FUNCTION_BLOCK "GCS7_E_FBAL"	// FB 28
TITLE = MZAG/MZAH/MZDE Flowbalancer
//  
//COPYRIGHT:    (C) 1997 BY  BUHLER AG, CH-9240 UZWIL  SWITZERLAND
//
//PRODUCT:      GCS7
//
//TITLE:        Element MZAG/MZAH/FBAL,MZDE (Profibus and Opto22)
//              (GCPROVB Revision 11)
//
//-------------------------------------------------------------------------
//
//IDENT:        AUTHOR:             DEPT:                      DATE:
//FB28.7.6      A. Egli             BASE                       30-Oct-2008
//              - StStopping -->StStopped : Check LCStep<=2
//FB28.7.5      A. Egli             BASE                       12-Jun-2008
//              - Disable Alarm26 if InRestdischarge=True
//FB28.7.4      A. Egli             BASE                       09-Apr-2008
//              Disable Alarm 18 Battery Low
//FB28.7.3      A. Egli             CT3                        08-Apr-2008
//              - Remove StStopping -->StStarting 
//              - StStopping -->StStopped : Check LCStep=1
//              - Filter.A34NoProduct and A37Empty catched until stopped
//FB28.7.2      A. Egli             CT3                        25-Mai-2007
//              - Overflow weight OutNotErasableWeight is 999'999'999 
//FB28.7.1      A.Egli              CT3                        01-Dec-2005
//              Parameter Upload Change DBD86-->DBD88
//FB28.7.0      A.Egli              CT3                        05-Jan-2005
//              Parameter Upload (uses DB10)
//FB28.6.0      A.Egli              CT3                        17-Aug-2004
//              MZDE: InRestdicharge
//FB28.5.3      A.Egli              CT3                        13-Apr-2004
//              MZDE: Reset "CmdNewJob"
//FB28.5.2      A.Egli              CT3                        17-Nov-2003
//              - Alarm 90: Fault Remote Control
//              - Ignor SumFault as long AlarmNr <> 0
//              - ComFault in mocal mode: change to StStopped 
//FB28.5.1      A. Egli             CT3                        11-Nov-2003
//              - No restart during StStopping.
//FB28.5.0      A. Egli             CT3                        09-Sep-2003
//              - ParMZDE 
//              - Condition for stoppen when stop point is reached 
//FB28.4.0      A. Egli             CT3                        17-Jun-2002
//              - New Release with one block 
//              - Profibus and Opto22 
//              - MZMN Micro Dosing
//              - LC Alarm 14 (DPFault) =Log Text number 12
//              - Command A: Command Flowrate in %
//FB28.3.1      A. Egli             CT3                        11-Jul-2000
//              MZAH mode: Command A, h
//FB28.3.0      A. Egli             CT3                        20-Jun-2000
//              Automatic set zero point
//FB28.2.2      A. Egli             CT3                        17-Mar-2000
//              Length for answer telegram
//FB33.2B       A. Egli             CT3                        20-Juli-1999
//              No fault is element InLocal
//FB33.2A       S. Kalberer         CT3                        11-Mar-1999
//              Correction factor ('K') included
//              CmdNewJob sets CmdNewValue
//FB33.1A       A. Egli             CT3                        16-Apr-1998
//              1st Release in S7
//
//-------------------------------------------------------------------------
//
//PURPOSE:      MANUAL : see [MZAHxxMAN]
//
//RESTRICTIONS: S7
//
//              (*2) : Not used for MZDE
//
//=======================================================
//Log Message: 
//------------------------------------------------------
//0     = Fault Cannceled
//1..79 = AlarmLC : Alarmnumber see manual of MEAF
//90    = Fault Remote Control
//91    = StStopped
//92    = StDosing
//93    = StEmptied
//94    = Timeout starting
//95    = Wrong value
//96    = Communication fault
//97    = 
//98    = 
//99    = Collected alarm
//
//=======================================================
//StCode:  State               
//------------------------------------------------------
//32    StFault                 
// 1    StStopped                   Stopped
//41    Stopped.HWStop              StStopped + InHWStop 
//51    Stopped.DPFault             StStopped + DPFault
// 2    StStarting              
// 3    StStarted               
// 7    StStopping              
//
//
AUTHOR : EA
FAMILY : GCS7LL
NAME : FBAL
VERSION : 7.6
VAR
  StCode : INT ;	//Element state code
  InEnable : BOOL ;	//Enable to run the element (manual and automatic mode)
  InRestdischarge : BOOL ;	//Rest discharge of the bin
  spare22 : BOOL ;
  CmdSetZeroPoint : BOOL ;	//Set zero point (*2)
  CmdNewValue : BOOL ;	//Send new target values
  CmdNewJob : BOOL ;	//Clear actual values (*2)
  CmdCorrFactor : BOOL ;	//Set correction factor (*2)
  tmpFilter34_37 : BOOL ;
  CmdOff : BOOL ;	//Pulse to stop the element (manual mode)
  CmdOn : BOOL ;	//Pulse to start the element (manual mode)
  CmdNext : BOOL ;	//Pulse to start the element in automatic mode
  CmdFaultReset : BOOL ;	//Command to reset fault
  InLocal : BOOL ;	//1= Local mode (no fault by start with service switch)
  InManual : BOOL ;	//1= Manual / 0= Automatic
  InReport : BOOL ;	//Report of all state transitions
  spare0307 : BOOL ;
  InHWStop : BOOL ;	//HW stop is detected, no fault
  InDPFault : BOOL ;	//DP-Fault is detected, no fault
  InSimulation : BOOL ;	//MZAH: Simulation with DPSim
  OutComFault : BOOL ;	//Communication fault
  OutBinEmpty : BOOL ;	//FBAL is rest discharged (*2)
  OutSetZeroPoint : BOOL ;	//(*2)
  OutSystemAdjust : BOOL ;	//(*2)
  OutpDosingEnable : BOOL ;	//Digital output dosing enable (only Opto22)
  StStopped : BOOL ;	//Element is stopped
  StStarting : BOOL ;	//Element is starting
  StStarted : BOOL ;	//Element is dosing
  StStopping : BOOL ;	//Element is stopping
  StFault : BOOL ;	//Element has a communication or device fault
  spare55 : BOOL ;
  spare56 : BOOL ;
  spare57 : BOOL ;
  OutStopPoint : BOOL ;	//Target weight reached (*2)
  OutWrongValue : BOOL ;	//Wrong nominal values, rejected by MEAF
  InFlowrate : DINT ;	//Flowrate target value [0.1%] or [kg/h] ! MZDE:Position [0.1%]
  InJobWeight : DINT ;	//MZAH: Is send to LC (*2)
  InRecipeNr : INT ;	//MZAH: Is send to LC (*2)
  InCorrFactor : DINT  := L#1000;	//Correction factor (1000: neutral value = no correction) (*2)
  OutFlowrate : DINT ;	//Is read from LC  FBAL:[kg/h]  ! MZDE:Position [0.1%]
  OutJobWeight : DINT ;	//Is calculated by element out of the not erasable weight  (*2)
  OutTotalWeight : DINT ;	//Is read from LC: de: Totalgewicht (*2)
  OutScaleWeight : DINT ;	//Is read from LC
  OutSetZeroTime : INT ;	//Actual time to set zero point (*2)
  OutRecipeNr : INT ;	//Is read from MEAF (*2)
  OutLCStep : INT ;	//Is read from MEAF
  OutAlarmNr : INT ;	//Is read from MEAF
  OutAlarmNrLog : INT ;	//Last textnumber send to log
  Par : STRUCT
   ParObjectNo : INT ;	//Is used for communication with PC, e.g. for message
   ParMsgType : INT ;	//Is used for message (translation of state)
   ParHornCode : INT ;	//Is used by horn module
   ParLogOff : BOOL ;	//Report is off
   ParManual : BOOL ;	//Manual mode wihout interlocking
   ParWithFlowratePc : BOOL ;	//Target flowrate in 0.1 %
   ParMZAH : BOOL ;	//MZAH Mode
   ParOpto22 : BOOL ;	//1=OPTO22 communication, 0=DP
   ParMZDE : BOOL ;	//MZDE ELement
   ParFilter : STRUCT 	//Filter to alarm 1=Ignore alarm
    SumFault : BOOL ;	//All: de: Sammelalarm
    A05_24VToLow : BOOL ;	//All:
    A07ADRange : BOOL ;
    A08ADCalibration : BOOL ;
    A09ADFunction : BOOL ;
    A10ADSupply : BOOL ;
    A11AnalogInput : BOOL ;
    AxxCommunication : BOOL ;	//A12: Serial Interface ; A14=DPFault
    A13RemoteControl : BOOL ;
    A16Printer : BOOL ;
    A24WeightHopper : BOOL ;
    A25FrequenceConverter : BOOL ;
    A26Tolerance : BOOL ;
    A27Measurment : BOOL ;
    A28Feeddrive : BOOL ;
    A29FeedingTime : BOOL ;
    A30ZeroTara : BOOL ;	//MZAH
    A32InletSlideGate : BOOL ;	//MZAH
    A33AirPressure : BOOL ;	//MZAH
    A34NoProduct : BOOL ;
    A37Empty : BOOL ;	//MZAH
    A38Slide : BOOL ;	//MZAH
    A39AirPressure : BOOL ;	//MZAH
    A54Relais : BOOL ;	//MZMN
   END_STRUCT ;
   ParComDB : INT ;	//OPTO22  : Communication DB
   ParLCIdx : INT ;	//OPTO22  : Index of data record
   ParLCAddr : INT ;	//OPTO22  : Address of LC
   ParIOByteNr : INT ;	//PROFIBUS: Address of first input and output byte
   ParMonTime : INT ;	//Monitoring time starting and stopping
   OutMonTime : INT ;	//Monitoring time starting and stopping
   OutNotErasableWeight : DINT  := L#-1;	//Is read from FBAL
   OutHelpFlags : STRUCT 	//Is sent to FBAL
    OutAlarmTimeOut : BOOL ;
    CmdNewValue : BOOL ;
    CmdFaultReset : BOOL ;
    CmdNewJob : BOOL ;
    OutFaultResetDone : BOOL ;
    OutTestNewAlarm : BOOL ;	//Aux. signal to retry fault message
    CmdCorrFactor : BOOL ;
    spare0007 : BOOL ;
    OutRelevantFault : BOOL ;
    OutNoAlarm : BOOL ;	//Alarmnumber 0 is read form LC
    OutFlagFaultResetDone : BOOL ;
    OutWeightCleared : BOOL ;	//Erasable weight is cleared
    OutComFaultRead : BOOL ;
    OutComFaultSend : BOOL ;
   END_STRUCT ;
   Command : STRUCT
    Start : BOOL ;	//de: Start
    ResetWtTotal : BOOL ;	//FBAL: de: Total löschen (*2)
    Restdischarge : BOOL ;	//MZDE: de: Restentleeren
    spare03 : BOOL ;
    spare04 : BOOL ;
    OverwriteLL : BOOL ;	//FBAL: de: Kein Alarm bei Leerstand (*2)
    spare06 : BOOL ;
    AcceptNewDataReady : BOOL ;	//FBAL: de: Quittierung neue Werte Bereit
    spare10 : BYTE ;
    spare20 : BYTE ;
    CommandReady : BOOL ;	//de: Steuersignale gültig
    SetZeroPoint : BOOL ;	//MZAG: de: MZAG (*2)
    spare32 : BOOL ;
    spare33 : BOOL ;
    spare34 : BOOL ;
    ResetAlarm : BOOL ;	//de: Alarm löschen
    NewSendData : BOOL ;	//de: Aenderung Sendedaten
    AcceptNewRcvData : BOOL ;	//de: Quittierung Aenderung Empfangsdatensatz
   END_STRUCT ;
   Status : STRUCT
    Operation : BOOL ;	//de: Betrieb
    WtTotalReached_InPos : BOOL ;	//de: Total erreicht  : MZDE: Slide in position
    RestdischargeDone : BOOL ;	//MZDE: de: Restentleeren ausgeführt
    spare03 : BOOL ;
    TotalReady : BOOL ;	//de: Total bereit (*2)
    Empty : BOOL ;	//de: Silo leer (*2)
    WtPulse : BOOL ;	//de: Gewichtsimpuls (*2)
    NewDataReady : BOOL ;	//de: Neue Werte Bereit
    AnalogMode : BOOL ;	//0/4-20mA set value  (*2)
    SetZeroPoint_Recipe1 : BOOL ;	//(*2)
    SystemAdjust_Recipe2 : BOOL ;	//(*2)
    spare20 : BYTE ;
    spare30 : BOOL ;
    spare31 : BOOL ;
    spare32 : BOOL ;
    RemoteControl : BOOL ;	//de: Sollwertvorgabe Remote
    WrongValue : BOOL ;	//de: Falscher Sollwert
    SumFault : BOOL ;	//de: Sammelalarm
    AcceptNewSendData : BOOL ;	//de: Quittierung Aenderung Sendedaten
    NewRcvData : BOOL ;	//de: Aenderung Empfangsdaten
   END_STRUCT ;
   OutComFlags : STRUCT 	//Flags for communication
    i_Done : BOOL ;
    d_Done : BOOL ;
    h_done : BOOL ;
    Q_Done : BOOL ;
    P_Done : BOOL ;
    S_Done : BOOL ;
    K_Done : BOOL ;
    A_Done : BOOL ;
   END_STRUCT ;
  END_STRUCT ;
END_VAR
VAR_TEMP
  tmpLOGvalue : WORD ;	//LOG value
  tmpCommand : INT ;
  tmpFBNO : INT ;	//Number of the actual FB
  tmpFault : BOOL ;
  tmpOff : BOOL ;
  tmpOn : BOOL ;
  tmpLocal : BOOL ;
  tmpLocalFault : BOOL ;
  tmpReport : BOOL ;
  tmpFlag : BOOL ;
  tmpOutLCAlarmBinEmpty : BOOL ;
  tmpLenDyn : DINT ;
  tmpWt : DINT ;
  tmpFilter : ARRAY  [0 .. 100 ] OF BOOL ;
  tmpComDB : INT ;
  tmpStatus_h : STRUCT 	//Is read from FBAL
   Remote : BOOL ;
   NewValue : BOOL ;
   Z1_Bit2 : BOOL ;
   BinEmpty : BOOL ;
   Z2_Bit0 : BOOL ;
   Z2_Bit1 : BOOL ;
   Z2_Bit2 : BOOL ;
   SumFault : BOOL ;
  END_STRUCT ;
  tmpStatus_i : STRUCT 	//Is read from FBAL
   EnableInactive : BOOL ;
   AlarmActive : BOOL ;
   AnalogMode : BOOL ;	//0/4-20mA set value
   SetZeroPoint : BOOL ;
   SystemAdjust : BOOL ;
   spare15 : BOOL ;	//only MEAF
   spare16 : BOOL ;	//only MEAF
   NominalFailure : BOOL ;	//Nominal value < 1%
  END_STRUCT ;
  tmpCommand_A : STRUCT
   Start : BOOL ;
   Stop : BOOL ;
   ResetWtTotal : BOOL ;
   AlarmReset : BOOL ;
   ValueInPc : BOOL ;
   Z3_1 : BOOL ;
   Z3_2 : BOOL ;
   Modify : BOOL ;
  END_STRUCT ;
  tmpCommand_S : STRUCT
   SetDosingRelease : BOOL ;
   AlarmReset : BOOL ;
   spare16 : BOOL ;
   SetZeroPoint : BOOL ;
   ClearPowerFlag : BOOL ;
   ResetWtTotal : BOOL ;
   spare12 : BOOL ;
   spare13 : BOOL ;
  END_STRUCT ;
  tmpAddr : WORD ;
  tmpReturn : INT ;
  DPData : STRUCT
   StatusCommand : DWORD ;
   NrSndDataSet : BYTE ;	//de: Nummer Sendedatensatz
   IdxSndDataSet : BYTE ;	//de: Index Sendedatensatz
   NrRcvDataSet : BYTE ;	//de: Nummer Empfangsdatensatz
   IdxRcvDataSet : BYTE ;	//de: Index Empfangsdatensatz
   Data : ARRAY  [1 .. 4 ] OF DINT ;
  END_STRUCT ;
  Set001 : STRUCT
   FlowrateAc : DINT ;	//de: Istleistung kg/h
   WtTotalAc : DINT ;	//de: Isttotalgewicht kg
   WtNotErasable : DINT ;	//de: nochtlöschbarese Totalgewicht
   spare12 : BYTE ;
   RecipeNr : BYTE ;
   Step : BYTE ;
   AlarmNr : BYTE ;
  END_STRUCT ;
END_VAR
BEGIN
NETWORK
TITLE =  Start Global
      L     28;
      T     #tmpFBNO;
      L     88;
      T     #tmpLenDyn;	//--> Len dynamic data in byte
      L     #Par.ParComDB;
      T     #tmpComDB;
NETWORK
TITLE = Filter
      LAR1  P##tmpFilter;
      L     0;
      T     LD [AR1,P#0.0];	//tmpFilter[00..31]  //[5.0]
      T     LD [AR1,P#4.0];	//tmpFilter[32..63]  //[5.0]
      T     LD [AR1,P#8.0];	//tmpFilter[64..95]  //[5.0]
      SET;	//[5.2]
      =     #tmpFilter[0];
      A     #Par.ParFilter.A05_24VToLow;
      =     #tmpFilter[5];
      A     #Par.ParFilter.A07ADRange;
      =     #tmpFilter[7];
      A     #Par.ParFilter.A08ADCalibration;
      =     #tmpFilter[8];
      A     #Par.ParFilter.A09ADFunction;
      =     #tmpFilter[9];
      A     #Par.ParFilter.A10ADSupply;
      =     #tmpFilter[10];
      A     #Par.ParFilter.A11AnalogInput;
      =     #tmpFilter[11];
      A     #Par.ParFilter.AxxCommunication;
      =     #tmpFilter[12];
      =     #tmpFilter[14];	//[1.4]
      A     #Par.ParFilter.A13RemoteControl;
      =     #tmpFilter[13];
      A     #Par.ParFilter.A16Printer;
      =     #tmpFilter[16];
      SET;
      =     #tmpFilter[18];	//[7.4] Battery Low
      A     #Par.ParFilter.A24WeightHopper;
      =     #tmpFilter[24];
      A     #Par.ParFilter.A25FrequenceConverter;
      =     #tmpFilter[25];
      A     #Par.ParFilter.A26Tolerance;
      O     #InRestdischarge;	//[7.5]
      =     #tmpFilter[26];
      A     #Par.ParFilter.A27Measurment;
      =     #tmpFilter[27];
      A     #Par.ParFilter.A28Feeddrive;
      =     #tmpFilter[28];
      A     #Par.ParFilter.A29FeedingTime;
      =     #tmpFilter[29];
      A     #Par.ParFilter.A30ZeroTara;
      =     #tmpFilter[30];
      A     #Par.ParFilter.A32InletSlideGate;
      =     #tmpFilter[32];
      A     #Par.ParFilter.A33AirPressure;
      =     #tmpFilter[33];
      A     #InRestdischarge;	//[7.3]
      S     #tmpFilter34_37;	//[7.3]
      A     #StStopped;	//[7.3]
      R     #tmpFilter34_37;	//[7.3]
      A     #tmpFilter34_37;	//[7.3]
      A     #StStopping;	//[7.3]
      O     #Par.ParFilter.A34NoProduct;
      O     #InRestdischarge;
      =     #tmpFilter[34];
      A     #tmpFilter34_37;	//[7.3]
      A     #StStopping;	//[7.3]
      O     #Par.ParFilter.A37Empty;
      O     #InRestdischarge;
      =     #tmpFilter[37];
      A     #Par.ParFilter.A38Slide;
      =     #tmpFilter[38];
      A     #Par.ParFilter.A39AirPressure;
      =     #tmpFilter[39];
      A     #Par.ParFilter.A54Relais;
      =     #tmpFilter[54];
NETWORK
TITLE = (Opto22) Call back function
//*****This functions are called by FBxxx (COM) ******
      AN    #Par.ParOpto22;
      JC    O22Z;
      OPN   DB [#tmpComDB];
      L     0;
      L     DBW 32;	//COM.Element.CODE;
      ==I;
      JC    PC;
      L     DBB 76;	//COM.Telegram.Command;
      T     #tmpCommand;
      L     1;
      L     DBW 32;	//COM.Element.CODE;
      ==I;
      JC    Send;
      L     2;
      ==I;
      JC    Rcv;
      L     4;	//NAK
      L     DBW 32;	//COM.Element.CODE;
      ==I;
      S     #OutComFault;	//fault communication
      JU    STOR;
//Read telegram length
Send: L     #tmpCommand;
      L     'd';
      ==I;
      L     16;	//Lenght in byte
      JC    Sndx;
      L     #tmpCommand;
      L     'i';
      ==I;
      L     6;	//Lenght in byte
      JC    Sndx;
      L     #tmpCommand;
      L     'h';
      ==I;
      L     36;	//Lenght in byte
      JC    Sndx;
      JU    SndW;
Sndx: T     DBW 86;	//COM.Telegram.LenAnswer
      JU    STOR;
SndW: NOP   0;
//======================================================================
//Prepare Send Data 
//======================================================================
//--------------------
//Send Q
//--------------------
      L     #tmpCommand;
      L     'Q';
      <>I;
      JC    SndP;
      L     #InFlowrate;
      T     DBD 36;	//COM.Element.InOutValue
      L     16;	//Convert DInt to 6-ASCII
      T     DBW 0;	//COM.CODE
      L     6;	//Lenght in byte
      JU    Snd1;
//--------------------
//Send P
//--------------------
SndP: L     #tmpCommand;
      L     'P';
      <>I;
      JC    SndK;
      L     #InFlowrate;
      T     DBD 36;	//COM.Element.InOutValue
      L     14;	//Convert DInt to 4-ASCII
      T     DBW 0;	//COM.CODE
      L     4;	//Lenght in byte
      JU    Snd1;
//--------------------
//Send K [2.A]
//--------------------
SndK: L     #tmpCommand;
      L     'K';
      <>I;
      JC    SndA;
      L     #InCorrFactor;
      T     DBD 36;	//COM.Element.InOutValue
      L     16;	//Convert DInt to 6-ASCII
      T     DBW 0;	//COM.CODE
      L     6;	//Lenght in byte
      JU    Snd1;
//--------------------
//Send A [3.1]
//--------------------
SndA: L     #tmpCommand;
      L     'A';
      <>I;
      JC    SndS;
      LAR1  P##tmpCommand_A;
      L     0;
      T     LW [AR1,P#0.0];	//-->Reset tmpStateTarget
//command 1
      A     #Par.Command.Start;
      =     #tmpCommand_A.Start;
      AN    #Par.Command.Start;
      =     #tmpCommand_A.Stop;
      A     #Par.Command.ResetWtTotal;
      =     #tmpCommand_A.ResetWtTotal;
      A     #Par.Command.ResetAlarm;
      =     #tmpCommand_A.AlarmReset;
      A     #Par.ParWithFlowratePc;	//[4.0]
      =     #tmpCommand_A.ValueInPc;	//[4.0]
      SET;
      =     #tmpCommand_A.Modify;
      L     0;	//Character offset
      T     DBW 40;	//COM.Element.AddrOffset
      LAR1  P##tmpCommand_A;
      L     LB [AR1,P#0.0];
      T     DBD 36;	//COM.Element.InOutValue
      L     31;	//Convert Hex to 1-ASCII
      T     DBW 0;	//COM.CODE
      CDB;	//ComDB->Instanz-DB
      UC    "GCS7_RS485Ctrl";	//Convert (CODE=DBW0)
      CDB;	//ElementDB->Instanz-DB
//n.b   
      L     1;	//Character offset
      T     DBW 40;	//COM.Element.AddrOffset
      L     0;
      T     DBD 36;	//COM.Element.InOutValue
      L     32;	//Convert Hex to 1-ASCII
      T     DBW 0;	//COM.CODE
      CDB;	//ComDB->Instanz-DB
      UC    "GCS7_RS485Ctrl";	//Convert (CODE=DBW0)
      CDB;	//ElementDB->Instanz-DB
// Command 2    
      L     3;	//Character offset
      T     DBW 40;	//COM.Element.AddrOffset
      LAR1  P##tmpCommand_A;
      L     LB [AR1,P#0.0];
      SRW   4;
      T     DBD 36;	//COM.Element.InOutValue
      L     31;	//Convert Hex to 1-ASCII
      T     DBW 0;	//COM.CODE
      CDB;	//ComDB->Instanz-DB
      UC    "GCS7_RS485Ctrl";	//Convert (CODE=DBW0)
      CDB;	//ElementDB->Instanz-DB
// n.b    
      L     4;	//Character offset
      T     DBW 40;	//COM.Element.AddrOffset
      L     0;
      T     DBD 36;	//COM.Element.InOutValue
      L     16;	//Convert DInt to 6-ASCII
      T     DBW 0;	//COM.CODE
      CDB;	//ComDB->Instanz-DB
      UC    "GCS7_RS485Ctrl";	//Convert (CODE=DBW0)
      CDB;	//ElementDB->Instanz-DB
// Flowrate    
      L     6;	//Character offset
      T     DBW 40;	//COM.Element.AddrOffset
      L     #InFlowrate;
      T     DBD 36;	//COM.Element.InOutValue
      L     16;	//Convert DInt to 6-ASCII
      T     DBW 0;	//COM.CODE
      CDB;	//ComDB->Instanz-DB
      UC    "GCS7_RS485Ctrl";	//Convert (CODE=DBW0)
      CDB;	//ElementDB->Instanz-DB
// InJobWeight                          //[5.0]
      L     12;	//Character offset
      T     DBW 40;	//COM.Element.AddrOffset
      L     #InJobWeight;
      T     DBD 36;	//COM.Element.InOutValue
      L     18;	//Convert DInt to 8-ASCII
      T     DBW 0;	//COM.CODE
      CDB;	//ComDB->Instanz-DB
      UC    "GCS7_RS485Ctrl";	//Convert (CODE=DBW0)
      CDB;	//ElementDB->Instanz-DB
      L     20;	//Lenght in byte
      T     DBW 78;	//COM.Telegram.Len
      JU    SndZ;
//--------------------
//Send S
//--------------------
SndS: L     #tmpCommand;
      L     'S';
      <>I;
      JC    SndZ;
      LAR1  P##tmpCommand_S;
      L     0;
      T     LW [AR1,P#0.0];	//-->Reset tmpStateTarget
      A     #Par.Command.Start;
      =     #tmpCommand_S.SetDosingRelease;
      A     #Par.Command.ResetAlarm;
      =     #tmpCommand_S.AlarmReset;
      =     #tmpCommand_S.ClearPowerFlag;
      A     #Par.Command.SetZeroPoint;
      =     #tmpCommand_S.SetZeroPoint;
      A     #Par.Command.ResetWtTotal;
      =     #tmpCommand_S.ResetWtTotal;
      LAR1  P##tmpCommand_S;
      L     LB [AR1,P#0.0];
      T     DBD 36;	//COM.Element.InOutValue
      L     32;	//Convert Hex to 2-ASCII
      T     DBW 0;	//COM.CODE
      L     2;	//Lenght in byte
Snd1: T     DBW 78;	//COM.Telegram.Len
      CDB;	//ComDB->Instanz-DB
      UC    "GCS7_RS485Ctrl";	//Convert (CODE=DBW0)
      CDB;	//ElementDB->Instanz-DB
SndZ: JU    STOR;
//======================================================================
//Answer Telegramm: Copy reveived data to element
//======================================================================
//--------------------
//Receive h 
//--------------------
Rcv:  R     #OutComFault;
      L     #tmpCommand;
      L     'h';
      <>I;
      JC    Rcvi;
      AN    #Par.OutHelpFlags.OutFaultResetDone;
      JC    r_H1;
      S     #Par.OutHelpFlags.OutTestNewAlarm;
//StepNr
r_H1: L     2;	//Character offset
      T     DBW 40;	//COM.Element.AddrOffset
      L     22;	//Convert 2-ASCII to DInt
      T     DBW 0;	//COM.CODE
      CDB;	//ComDB->Instanz-DB
      UC    "GCS7_RS485Ctrl";	//Convert (CODE=DBW0)
      CDB;	//ElementDB->Instanz-DB
      L     DBD 36;	//COM.Element.InOutValue
      T     #OutLCStep;
//LC status
      L     0;	//Character offset
      T     DBW 40;	//COM.Element.AddrOffset
      L     42;	//Convert 2-ASCII to Hex
      T     DBW 0;	//COM.CODE
      CDB;	//ComDB->Instanz-DB
      UC    "GCS7_RS485Ctrl";	//Convert (CODE=DBW0)
      CDB;	//ElementDB->Instanz-DB
      L     DBD 36;	//COM.Element.InOutValue
      LAR1  P##tmpStatus_h;
      T     LB [AR1,P#0.0];	//-->tmpStatus_h
      A     #tmpStatus_h.Remote;
      =     #Par.Status.RemoteControl;
      A     #tmpStatus_h.BinEmpty;
      =     #Par.Status.Empty;
      A     #tmpStatus_h.SumFault;
      =     #Par.Status.SumFault;
      L     #OutLCStep;
      L     3;
      >=I;
      =     #Par.Status.Operation;
      L     2;
      L     #OutLCStep;
      ==I;
      =     #Par.Status.SetZeroPoint_Recipe1;
//Alarm number / LC alarm bit mask
      L     4;	//Character offset
      T     DBW 40;	//COM.Element.AddrOffset
      L     22;	//Convert 2-ASCII to DInt
      T     DBW 0;	//COM.CODE
      CDB;	//ComDB->Instanz-DB
      UC    "GCS7_RS485Ctrl";	//Convert (CODE=DBW0)
      CDB;	//ElementDB->Instanz-DB
      L     DBD 36;	//COM.Element.InOutValue
      T     #OutAlarmNr;
//Filter SumFault
      L     #OutAlarmNr;	//[5.2]
      L     0;	//[5.2]
      <>I;	//[5.2]
      O     #Par.ParFilter.SumFault;	//[5.2]
      O     #InRestdischarge;	//[5.2]
      =     #tmpFilter[0];	//[5.2]
//Acutal flowrate
      L     6;	//Character offset
      T     DBW 40;	//COM.Element.AddrOffset
      L     26;	//Convert 6-ASCII to DInt
      T     DBW 0;	//COM.CODE
      CDB;	//ComDB->Instanz-DB
      UC    "GCS7_RS485Ctrl";	//Convert (CODE=DBW0)
      CDB;	//ElementDB->Instanz-DB
      L     DBD 36;	//COM.Element.InOutValue
      T     #OutFlowrate;
//ScaleWeight
      L     12;	//Character offset
      T     DBW 40;	//COM.Element.AddrOffset
      L     26;	//Convert 6-ASCII to DInt
      T     DBW 0;	//ERH.CODE
      CDB;	//ComDB->Instanz-DB
      UC    "GCS7_RS485Ctrl";	//Convert (CODE=DBW0)
      CDB;	//ElementDB->Instanz-DB
      L     DBD 36;	//ERH.Element.InOutValue
      T     #OutScaleWeight;	//[4.0]
//- OutErasableWeight
      L     18;	//Character offset
      T     DBW 40;	//ERH.Element.AddrOffset
      L     28;	//Convert 8-ASCII to DInt
      T     DBW 0;	//ERH.CODE
      CDB;	//ComDB->Instanz-DB
      UC    "GCS7_RS485Ctrl";	//Convert (CODE=DBW0)
      CDB;	//ElementDB->Instanz-DB
      L     DBD 36;	//ERH.Element.InOutValue
      T     #OutTotalWeight;	//[4.0]
//Not erasable total
      L     26;	//Character offset
      T     DBW 40;	//COM.Element.AddrOffset
      L     28;	//Convert 8-ASCII to DInt
      T     DBW 0;	//COM.CODE
      CDB;	//ComDB->Instanz-DB
      UC    "GCS7_RS485Ctrl";	//Convert (CODE=DBW0)
      CDB;	//ElementDB->Instanz-DB
      L     DBD 36;	//COM.Element.InOutValue
      T     #tmpWt;
      JU    RdJ1;
//--------------------
//Receive i 
//--------------------
Rcvi: R     #OutComFault;
      L     #tmpCommand;
      L     'i';
      <>I;
      JC    Rcvd;
      AN    #Par.OutHelpFlags.OutFaultResetDone;
      JC    r_J1;
      S     #Par.OutHelpFlags.OutTestNewAlarm;
//LC status
r_J1: L     2;	//Character offset
      T     DBW 40;	//COM.Element.AddrOffset
      L     42;	//Convert 2-ASCII to Hex
      T     DBW 0;	//COM.CODE
      CDB;	//ComDB->Instanz-DB
      UC    "GCS7_RS485Ctrl";	//Convert (CODE=DBW0)
      CDB;	//ElementDB->Instanz-DB
      L     DBD 36;	//COM.Element.InOutValue
      LAR1  P##tmpStatus_i;
      T     LB [AR1,P#0.0];
      AN    #tmpStatus_i.EnableInactive;
      =     #Par.Status.Operation;
      A     #tmpStatus_i.AlarmActive;
      =     #Par.Status.SumFault;
      A     #tmpStatus_i.AnalogMode;
      =     #Par.Status.AnalogMode;
      A     #tmpStatus_i.SetZeroPoint;
      =     #Par.Status.SetZeroPoint_Recipe1;
      A     #tmpStatus_i.SystemAdjust;
      =     #Par.Status.SystemAdjust_Recipe2;
      A     #tmpStatus_i.NominalFailure;
      =     #Par.Status.WrongValue;
//Alarm number / LC alarm bit mask
      L     4;	//Character offset
      T     DBW 40;	//COM.Element.AddrOffset
      L     22;	//Convert 2-ASCII to DInt
      T     DBW 0;	//COM.CODE
      CDB;	//ComDB->Instanz-DB
      UC    "GCS7_RS485Ctrl";	//Convert (CODE=DBW0)
      CDB;	//ElementDB->Instanz-DB
      L     DBD 36;	//COM.Element.InOutValue
      T     #OutAlarmNr;
//  Convert AlarmNr to MEAF-MZAH
//    --------------
      L     1;	//Ram defective
      L     #OutAlarmNr;
      ==I;
      L     2;	//--> MEAF: RAM
      JC    riAL;
//    --------------
      L     2;	//Ram Battery
      L     #OutAlarmNr;
      ==I;
      L     6;	//--> MEAF: Data lost
      JC    riAL;
//    --------------
      L     3;	//Eprom
      L     #OutAlarmNr;
      ==I;
      L     1;	//--> MEAF: Eprom
      JC    riAL;
//    --------------
      L     4;	//24V
      L     #OutAlarmNr;
      ==I;
      L     5;	//--> MEAF: 24V
      JC    riAL;
//    --------------
      L     5;	//Trap
      L     #OutAlarmNr;
      ==I;
      L     3;	//--> MEAF: Runtime error Software
      JC    riAL;
//    --------------
      L     6;	//24V output Overload
      L     #OutAlarmNr;
      ==I;
      L     5;	//--> MEAF: 24V
      JC    riAL;
//    --------------
      L     8;	//Serial interface
      L     #OutAlarmNr;
      ==I;
      L     12;	//--> MEAF:Timemout Host
      JC    riAL;
//    --------------
      L     9;	//Bin Low Level
      L     #OutAlarmNr;
      ==I;
      L     37;	//--> MEAF:Timemout Host
      JC    riAL;
      L     #OutAlarmNr;	//ELSE
riAL: T     #OutAlarmNr;
      L     #OutAlarmNr;
      L     37;
      ==I;
      =     #Par.Status.Empty;
      JU    STOR;
//--------------------
// Receive 'd'
//--------------------
Rcvd: L     #tmpCommand;
      L     'd';
      <>I;
      JC    RcvS;
//Acutal flowrate
      L     0;	//Character offset
      T     DBW 40;	//COM.Element.AddrOffset
      L     26;	//Convert 6-ASCII to DInt
      T     DBW 0;	//COM.CODE
      CDB;	//ComDB->Instanz-DB
      UC    "GCS7_RS485Ctrl";	//Convert (CODE=DBW0)
      CDB;	//ElementDB->Instanz-DB
      L     DBD 36;	//COM.Element.InOutValue
      T     #OutFlowrate;
//Not erasable total
      L     6;	//Character offset
      T     DBW 40;	//COM.Element.AddrOffset
      L     28;	//Convert 8-ASCII to DInt
      T     DBW 0;	//COM.CODE
      CDB;	//ComDB->Instanz-DB
      UC    "GCS7_RS485Ctrl";	//Convert (CODE=DBW0)
      CDB;	//ElementDB->Instanz-DB
      L     DBD 36;	//COM.Element.InOutValue
      T     #tmpWt;
//---  Init first, if old value < 0  ---
RdJ1: L     #Par.OutNotErasableWeight;
      L     0;
      <D;
      JC    rgZ2;
//---  Calculate Weight ---
      L     #tmpWt;
      L     #Par.OutNotErasableWeight;
      -D;
      JM    rgZ1;
      JU    rgPo;
rgZ1: L     L#100000000;
      +D;
rgPo: L     10000;	// Maximum change by relaod software
      >D;
      JC    rgZ2;
      TAK;
      L     #OutJobWeight;
      +D;
      T     #OutJobWeight;	//--> Total weight
rgZ2: L     #tmpWt;
      T     #Par.OutNotErasableWeight;
      JU    STOR;
//--------------------
//Accept 'S','A'
//--------------------
RcvS: L     #tmpCommand;
      L     'S';
      <>I;
      A(;
      L     #tmpCommand;
      L     'A';
      <>I;
      );
      JC    RcvP;
      AN    #Par.Command.ResetAlarm;
      JC    tS1;
      S     #Par.OutHelpFlags.OutFaultResetDone;
tS1:  SET;
      R     #Par.OutHelpFlags.CmdNewJob;
      R     #Par.OutHelpFlags.CmdFaultReset;
      R     #Par.Command.ResetAlarm;
      R     #Par.Command.ResetWtTotal;
      R     #Par.OutHelpFlags.CmdNewValue;
      AN    #Par.Command.SetZeroPoint;
      JC    STOR;	//[3.0]
      R     #Par.Command.SetZeroPoint;	//[3.0]
      L     0;	//[3.0]
      T     #OutSetZeroTime;	//[3.0]
      JU    STOR;
RcvP: L     #tmpCommand;
      L     'P';
      <>I;
      JC    RcvQ;
      R     #Par.OutHelpFlags.CmdNewValue;
      JU    STOR;
RcvQ: L     #tmpCommand;
      L     'Q';
      <>I;
      JC    RcvK;
      R     #Par.OutHelpFlags.CmdNewValue;
//--------------------
//Accept 'K'
//--------------------
RcvK: L     #tmpCommand;
      L     'K';
      <>I;
      JC    RcvX;
      R     #Par.OutHelpFlags.CmdCorrFactor;
RcvX: JU    STOR;
O22Z: NOP   0;
NETWORK
TITLE = PC Control
//=== Test Object number =====================
PC:   L     "SYS_DirectCtrlDB".PC.ObjectNo;	//PCControl.ObjectNo
      L     #Par.ParObjectNo;	//Input ObjectNo
      <>I;
      JC    Ctrl;
//=== Test OType      ========================
      L     1028;	//Input object type
      L     "SYS_DirectCtrlDB".PC.ObjectType;	//PCControl.ObjectType
      <>I;
      JC    Ctrl;
//=== Test Handshake =========================
      A     "SYS_DirectCtrlDB".PC.Hsk.FExamine;	//Handshake.FExamine
      JC    pExa;
      A     "SYS_DirectCtrlDB".PC.Hsk.FDefineCmd;	//Handshake.FDefineCmd
      JC    pCmd;
      A     "SYS_DirectCtrlDB".PC.Hsk.FDefinePara;	//Handshake.FDefinePara
      JC    pPar;
pIni: L     2;	//FcInit
      UC    "SYS_DirectCtrl";
      JU    Ctrl;
//Write parameter 
pPar: NOP   0;
//Write new commands from PC to Interface of group 
pCmd: A     "SYS_DirectCtrlDB".PC.Cmd1[1];	//Cmd1[1]  =CmdRestDischargeOn
      S     #InRestdischarge;
      A     "SYS_DirectCtrlDB".PC.Cmd2[1];	//Cmd1[2]  =CmdRestDischargeOff
      R     #InRestdischarge;
      A     "SYS_DirectCtrlDB".PC.Cmd1[3];	//Cmd1[4]  =CmdSetZeroPoint
      S     #CmdSetZeroPoint;
      A     "SYS_DirectCtrlDB".PC.Cmd1[4];	//Cmd1[4]  =CmdNewValue
      S     #CmdNewValue;
      A     "SYS_DirectCtrlDB".PC.Cmd1[5];	//Cmd1[5]  =CmdNewJob
      S     #CmdNewJob;
      A     "SYS_DirectCtrlDB".PC.Cmd1[6];	//Cmd1[6]  =CmdCorrFactor
      S     #CmdCorrFactor;
      A     "SYS_DirectCtrlDB".PC.Cmd1[8];	//Cmd1[8]  =CmdOff
      S     #CmdOff;
      A     "SYS_DirectCtrlDB".PC.Cmd1[9];	//Cmd1[9]  =CmdOn
      S     #CmdOn;
      A     "SYS_DirectCtrlDB".PC.Cmd1[10];	//Cmd1[10] =CmdNext
      S     #CmdNext;
      A     "SYS_DirectCtrlDB".PC.Cmd1[11];	//Cmd1[11] =CmdFaultReset
      S     #CmdFaultReset;
      A     "SYS_DirectCtrlDB".PC.Cmd1[13];	//Cmd1[13] =CmdManualOn
      S     #InManual;
      A     "SYS_DirectCtrlDB".PC.Cmd2[13];	//Cmd2[13] =CmdManualOff
      R     #InManual;
      A     "SYS_DirectCtrlDB".PC.Cmd1[14];	//Cmd1[14] =CmdReportOn
      S     #InReport;
      A     "SYS_DirectCtrlDB".PC.Cmd2[14];	//Cmd2[14] =CmdReportOff
      R     #InReport;
//Define Value
      AN    "SYS_DirectCtrlDB".PC.Hsk.FDefineValue;	// PC.Hsk.FDefineValue
      ON    #InManual;
      JC    pIni;
      LAR1  P#DBX 58.0;
      L     DBD [AR1,P#8.0];
      T     #InFlowrate;
      L     DBD [AR1,P#12.0];
      T     #InJobWeight;
      L     DBW [AR1,P#16.0];
      T     #InRecipeNr;
      L     DBD [AR1,P#18.0];
      T     #InCorrFactor;
      JU    pIni;
pExa: TAR2;	//Address dynamic datas
      T     "SYS_DirectCtrlDB".GC.InDynAddr;	//-->PCControl.GC.InDynAddr
      L     #tmpLenDyn;	//Length dynamic datas
      T     "SYS_DirectCtrlDB".GC.InDynLen;	//-->PCControl.GC.InDynLen
      L     0;
      T     "SYS_DirectCtrlDB".GC.InParaAddr;	//-->PCControl.GC.InParaAddr
      T     "SYS_DirectCtrlDB".GC.InParaLen;	//-->PCControl.GC.InParaLen
      L     1;	//Code FcExamine
      UC    "SYS_DirectCtrl";
      L     11;	//Revision
      T     "SYS_DirectCtrlDB".GC.Revision;
Ctrl: NOP   0;
NETWORK
TITLE = [7.0] LCParameter
      L     #Par.ParObjectNo;
      L     "SYS_DirectCtrlLCDB".PC.ObjectNo;
      <>I;
      ON    #Par.ParOpto22;
      JC    LCP0;
      T     "SYS_DirectCtrlLCDB".GC.InObjectNo;
      L     #Par.ParComDB;
      T     "SYS_DirectCtrlLCDB".GC.InDBNr;
      L     #Par.ParLCAddr;
      T     "SYS_DirectCtrlLCDB".GC.InLCAddr;
LCP0: NOP   0;
NETWORK
TITLE =  Read LC data
      AN    #Par.ParOpto22;
      JC    O22A;
      OPN   DB [#tmpComDB];
      L     #Par.ParLCIdx;
      T     DBW 34;	//COM.Element.Index;
      L     1;	//Read LC data
      T     DBW 0;	//COM.CODE;
      CDB;
      UC    "GCS7_RS485Ctrl";
      CDB;
      L     #tmpFBNO;
      T     DBW 52;	//COM.LC0.FBNO;
      L     DINO;
      T     DBW 54;	//COM.LC0.DINO;
      TAR2  DBD 56;	//COM.LC0.AddrDyn;        
      L     0;
      T     DBD 60;	//COM.LC0.AddrPara;       
      L     #Par.ParLCAddr;
      T     DBD 64;	//COM.Telegram.LCAddr;
O22A: NOP   0;
NETWORK
TITLE = (Profibus) Read data and store Data 
      A     #Par.ParOpto22;
      JC    DP_A;
      L     #Par.ParIOByteNr;
      T     #tmpAddr;
      A     #InSimulation;
      JC    rSim;
      CALL  "SIEMENS_DPRD_DAT" (
           LADDR                    := #tmpAddr,
           RET_VAL                  := #tmpReturn,
           RECORD                   := #DPData);
      L     #tmpReturn;
      L     0;
      <>I;
      =     #Par.OutHelpFlags.OutComFaultRead;
      JC    rcv0;
      JU    rDP;
//read from Simulation
rSim: R     #Par.OutHelpFlags.OutComFaultRead;
      A     "GCS7_Gr_SimDPtoImage";
      L     P#I 0.0;
      JC    rDB1;
      OPN   "TEST_IOSimuliInput";
      L     P#DBX 0.0;
rDB1: L     #Par.ParIOByteNr;
      SLD   3;
      +D;
      LAR1;
      L     D [AR1,P#0.0];
      T     #DPData.StatusCommand;
      L     B [AR1,P#4.0];
      T     #DPData.NrSndDataSet;
      L     B [AR1,P#5.0];
      T     #DPData.IdxSndDataSet;
      L     B [AR1,P#6.0];
      T     #DPData.NrRcvDataSet;
      L     B [AR1,P#7.0];
      T     #DPData.IdxRcvDataSet;
      L     D [AR1,P#8.0];
      T     #DPData.Data[1];
      L     D [AR1,P#12.0];
      T     #DPData.Data[2];
      L     D [AR1,P#16.0];
      T     #DPData.Data[3];
      L     D [AR1,P#20.0];
      T     #DPData.Data[4];
//==Copy Status===============
rDP:  L     #DPData.NrRcvDataSet;
      L     0;
      ==I;
      JC    R001;
      CALL  "SIEMENS_BLKMOV" (
           SRCBLK                   := #DPData.StatusCommand,
           RET_VAL                  := #tmpReturn,
           DSTBLK                   := #Par.Status);
      AN    #Par.Status.NewRcvData;
      A     #InSimulation;
      JC    rcv0;
//===============================
//Answer Dataset 001
      L     #DPData.NrRcvDataSet;
      L     1;
      <>I;
      JC    r11;	//[7.0]
      CALL  "SIEMENS_BLKMOV" (
           SRCBLK                   := #DPData.Data,
           RET_VAL                  := #tmpReturn,
           DSTBLK                   := #Set001);
      AN    #Par.ParMZDE;	//[5.0]
      JC    r1D1;	//[5.0]
      L     #Set001.FlowrateAc;	//[5.0]
      SRD   16;	//[5.0]
      T     #OutFlowrate;	//[5.0]
      JU    r1D2;	//[5.0]
r1D1: L     #Set001.FlowrateAc;
      T     #OutFlowrate;
      L     #Set001.WtTotalAc;
      T     #OutTotalWeight;
      L     #Set001.RecipeNr;
      T     #OutRecipeNr;
r1D2: L     #Set001.Step;
      T     #OutLCStep;
//Filter SumFault
      L     #Set001.AlarmNr;	//[5.2]
      L     0;	//[5.2]
      <>I;	//[5.2]
      O     #Par.ParFilter.SumFault;	//[5.2]
      O     #InRestdischarge;	//[5.2]
      =     #tmpFilter[0];	//[5.2]
//Reset old alarm flags with CmdFaultReset
      A     #Par.OutHelpFlags.OutFlagFaultResetDone;
      A     "SYS_Pulse1000ms";
      R     #Par.OutHelpFlags.OutFlagFaultResetDone;
      R     #Par.OutHelpFlags.OutFaultResetDone;
      S     #Par.OutHelpFlags.OutTestNewAlarm;
      L     0;
      L     #Set001.AlarmNr;
      ==I;
      =     #Par.OutHelpFlags.OutNoAlarm;
//  keep old alalrm number
      A     #Par.OutHelpFlags.OutNoAlarm;
      A     #Par.OutHelpFlags.OutRelevantFault;
      AN    #Par.OutHelpFlags.OutTestNewAlarm;
      AN    #InLocal;
      AN    #InManual;
      JC    rA1;
      T     #OutAlarmNr;
//--------------------------------------
//Calculate job weight on WtNotErasable
rA1:  L     #Set001.WtNotErasable;
//---  Init first, if old value < 0  ---
      L     #Par.OutNotErasableWeight;
      L     0;
      <D;
      JC    rtZ2;
//---  Calculate Weight ---
      L     #Set001.WtNotErasable;
      L     #Par.OutNotErasableWeight;
      -D;
      JM    rtZ1;
      JU    rtPo;
rtZ1: L     L#1000000000;	//[7.2] Overflow weight is 999'999'999
      +D;
      JM    rtZ2;	//[7.2]
rtPo: L     10000;	// Maximum change by relaod software
      >D;
      JC    rtZ2;
      TAK;
      L     #OutJobWeight;
      +D;
      T     #OutJobWeight;	//--> Total weight
rtZ2: L     #Set001.WtNotErasable;
      T     #Par.OutNotErasableWeight;
      JU    R11;	//[7.0]   
//===============================
//[7.0]--> LC Parameter 
//Reading dataset 11
R11:  L     "SYS_DirectCtrlLCDB".PC.ObjectNo;
      L     #Par.ParObjectNo;
      <>I;
      JC    R127;
      AN    "SYS_DirectCtrlLCDB".PC.Hsk.FExamineFirst;
      AN    "SYS_DirectCtrlLCDB".PC.Hsk.FExamineNext;
      JC    R127;
// -- Start Reading with Dataset 11
      L     11;
      T     #DPData.NrRcvDataSet;
      L     253;	//First
      A     "SYS_DirectCtrlLCDB".PC.Hsk.FExamineFirst;
      JC    rLC9;
      L     254;	//Next
rLC9: T     #DPData.IdxRcvDataSet;
      JU    rcv0;
//---Answer  dataset 11 ---
//---Answer  dataset 12 ---
r11:  L     #DPData.NrRcvDataSet;
      L     11;
      <>I;
      JC    rLCB;
// Answer Dataset 11
      L     '  ';
      T     "SYS_DirectCtrlLCDB".PC.Value[1];
      L     #DPData.Data[1];
      T     DB10.DBD 60;
      L     #DPData.Data[2];
      T     DB10.DBD 64;
      L     #DPData.Data[3];
      T     DB10.DBD 68;
      L     #DPData.Data[4];
      T     DB10.DBD 72;
      L     #DPData.IdxRcvDataSet;
      L     255;
      ==I;
      JC    rLCE;
      S     "SYS_DirectCtrlLCDB".GC.Set11Done;
      L     12;
      T     #DPData.NrRcvDataSet;
      L     0;
      T     #DPData.IdxRcvDataSet;
      JU    rcv0;	//--> Read dataset 12
// Answer Dataset 12
rLCB: L     #DPData.NrRcvDataSet;
      L     12;
      <>I;
      JC    r127;
      L     #DPData.Data[1];
      T     DB10.DBD 76;
      L     #DPData.Data[2];
      T     DB10.DBD 80;
      L     #DPData.Data[3];
      T     DB10.DBD 84;
      L     #DPData.Data[4];
      T     DB10.DBD 88;
      AN    "SYS_DirectCtrlLCDB".GC.Set11Done;
      JC    R127;
rLCE: L     12;
      CALL  "SYS_DirectCtrl";
      JU    R127;
//<--[7.0]
//===============================
//Answer  dataset 127
r127: L     #DPData.NrRcvDataSet;
      L     127;
      <>I;
      JC    r128;
      L     #DPData.Data[1];	//WtActual
      T     #OutScaleWeight;
      JU    R128;
//===============================
//Answer  dataset 128
r128: JU    r136;
//===============================
//Answer  dataset 136
r136: L     #DPData.NrRcvDataSet;
      L     136;
      <>I;
      JC    R001;	// =no valide answer read dataset 001
      JU    R001;
//===============================
//Read Dataset 001
R001: L     1;
      T     #DPData.NrRcvDataSet;
      L     0;
      T     #DPData.IdxRcvDataSet;
      A     #Par.OutHelpFlags.OutFaultResetDone;
      AN    "SYS_Pulse1000ms";
      S     #Par.OutHelpFlags.OutFlagFaultResetDone;
      JU    rcv0;
//===============================
//Read Dataset 127
R127: L     127;
      T     #DPData.NrRcvDataSet;
      L     0;
      T     #DPData.IdxRcvDataSet;
      JU    rcv0;
//===============================
//Read Dataset 128
R128: JU    R136;
//===============================
//Read Dataset 136
R136: JU    R001;
      JU    rcv0;
//===============================
rcv0: NOP   0;
DP_A: NOP   0;
NETWORK
TITLE = (Profibus) Status to ASW
      A     #Par.ParOpto22;
      JC    DP_E;
      A     #Par.OutHelpFlags.OutComFaultRead;
      O     #Par.OutHelpFlags.OutComFaultSend;
      =     #OutComFault;
//=======================================
//OutStopPoint 
//=======================================
      L     #OutJobWeight;
      L     #InJobWeight;
      >=D;
      A(;
      L     #InJobWeight;
      L     0;
      >D;	//[4.0]
      );
      O     #Par.Status.WtTotalReached_InPos;
      AN    #Par.OutHelpFlags.CmdNewJob;
      A(;
      AN    #Par.Command.ResetWtTotal;
      O     #InRestdischarge;
      );
      AN    #Par.ParMZDE;	//[5.0]
      =     #OutStopPoint;
//=======================================
//Init in local mode  
//=======================================
      AN    #InLocal;
      AN    #InManual;
      ON    #OutComFault;
      JC    alJL;
      L     0;
      T     #OutFlowrate;
alJL: NOP   0;
DP_E: NOP   0;
NETWORK
TITLE =  All State Init
//===Clear tmp Variable
//===Global Group Orders===
      A     "GCS7_Gr_OutManualOn";	//Global.OutManualOn
      S     #InManual;
      A     "GCS7_Gr_OutManualOff";	//Global.OutManualOff
      R     #InManual;
      A     #InManual;
      S     "GCS7_Gr_InManual";	//Global.InManualMode
//---Report is on---
      O     "GCS7_Gr_OutReportAll";	//---Global OutReportAll
      O     #InReport;
      =     #tmpReport;
//---FaultReset is on---
      A     "GCS7_Gr_OutFaultReset";	//Gr.OutFaultReset
      S     #CmdFaultReset;
//---State---
      A     #Par.Status.SetZeroPoint_Recipe1;	//[3.0]   
      AN    #Par.ParMZDE;	//[5.0]
      FP    #OutSetZeroPoint;	//[3.0]
      JCN   InZP;	//[3.0]
      L     3000;	//[3.0]
      T     #Par.OutMonTime;	//[3.0]
InZP: A     #Par.Status.SystemAdjust_Recipe2;
      AN    #Par.ParMZDE;	//[5.0]
      =     #OutSystemAdjust;
//---Local---
      A     #InLocal;
      AN    #InManual;
      =     #tmpLocalFault;
      A     #tmpLocalFault;
      O     #InHWStop;
      O     #InDPFault;
      =     #tmpLocal;
//---Off---
      AN    #InManual;
      ON    #Par.ParManual;
      AN    #InEnable;
      O     #tmpLocal;
      O     #CmdOff;
      O     #OutSetZeroPoint;
      O     #OutSystemAdjust;
      =     #tmpOff;
//---On---
      A     #CmdNext;
      AN    #InManual;
      O     #CmdOn;
      AN    #tmpOff;
      =     #tmpOn;
//--- Send Recipe
//--- Read Recipe
//--- tmpFault   
// Time out
      AN    #StStarting;
      AN    #StStopping;
      AN    #StFault;
      AN    #OutSetZeroPoint;
      R     #Par.OutHelpFlags.OutAlarmTimeOut;
      JC    inJ1;
      A     #Par.OutHelpFlags.OutAlarmTimeOut;
      O     #StFault;
      JC    inJ1;
      L     0;
      L     #Par.OutMonTime;
      >I;
      =     #Par.OutHelpFlags.OutAlarmTimeOut;
      AN    "GCS7_Gr_OutTick200ms";	// Global Tick 200ms
      JC    inJ1;
      +     -2;	// Decrement all 200ms
      T     #Par.OutMonTime;
inJ1: NOP   0;
//=======================================
//OutBinEmpty
//=======================================
      L     #OutAlarmNr;
      L     37;
      ==I;
      O     #Par.Status.Empty;
      AN    #Par.ParMZDE;	//[6.0]
      O;
      A     #Par.ParMZDE;	//[6.0]
      A     #Par.Status.RestdischargeDone;	//[6.0]
      S     #OutBinEmpty;	//[6.0]
      A     #Par.Status.Operation;
      AN    #Par.Status.Empty;
      AN    #Par.ParMZDE;	//[6.0]
      ON    #InRestdischarge;
      R     #OutBinEmpty;
//=======================================
//Fault   
//=======================================
      LAR1  P##tmpFilter;
      L     #OutAlarmNr;
      +AR1;	//Pointer to #tmpFilter[OutAlarmNumber]
      L     #OutAlarmNr;
      L     0;
      <>I;
      AN    L [AR1,P#0.0];	//#tmpFilter[OutAlarmNumber]
      O;
      A     #Par.Status.SumFault;
      AN    #tmpFilter[0];
      =     #Par.OutHelpFlags.OutRelevantFault;
      A     #Par.Status.WrongValue;
      =     #OutWrongValue;
      A     #Par.OutHelpFlags.OutRelevantFault;
      O     #OutComFault;
      O     #Par.OutHelpFlags.OutAlarmTimeOut;
      O     #Par.Status.WrongValue;
      O(;	//[5.2]
      AN    #Par.Status.RemoteControl;	//[5.2]
      AN    #Par.ParOpto22;	//[5.2]
      );	//[5.2]
      AN    #tmpLocal;
      =     #tmpFault;
//--- New Job
      A     #CmdNewJob;
      JCN   inEn;
      S     #CmdNewValue;	//2A:
      L     0;
      T     #OutJobWeight;	//--> Total weight
inEn: NOP   0;
//================================     //[5.0] Moved
      A     #Par.Command.Start;
      =     #tmpFlag;
      A     #tmpOn;
      AN    #Par.OutHelpFlags.CmdNewJob;
      AN    #Par.OutHelpFlags.CmdNewValue;
      S     #Par.Command.Start;
      A     #StFault;
      A     #Par.OutHelpFlags.OutNoAlarm;
      O     #Par.OutHelpFlags.CmdNewJob;
      O     #tmpOff;
      O;	//[2.3]
      A     #InRestdischarge;	//[2.3]
      A     #OutBinEmpty;	//[2.3]
      A     #StStopped;	//[2.3]
      AN    #Par.ParMZDE;	//[5.0]
      O     #StStopping;	//[5.1]
      R     #Par.Command.Start;
//================================
NETWORK
TITLE = (Profibus) Prepare Command for MEAF
      A     #Par.ParOpto22;
      JC    DP_B;
      A     #CmdNewJob;
      R     #CmdNewJob;
      S     #Par.OutHelpFlags.CmdNewJob;
//==============================
      A     #Par.Status.AcceptNewSendData;
      A     #Par.Command.ResetAlarm;
      R     #Par.Command.ResetAlarm;
      S     #Par.OutHelpFlags.OutFaultResetDone;
      A     #CmdFaultReset;
      AN    #Par.Status.AcceptNewSendData;
      R     #CmdFaultReset;
      S     #Par.Command.ResetAlarm;
      R     #Par.OutHelpFlags.OutAlarmTimeOut;
//================================
      A     #Par.Status.AcceptNewSendData;
      A     #Par.Command.ResetWtTotal;
      O;
      A     #Par.ParMZDE;	//[5.3]
      A     #Par.OutHelpFlags.CmdNewJob;	//[5.3]
      S     #Par.OutHelpFlags.OutWeightCleared;
      R     #Par.Command.ResetWtTotal;
      R     #Par.OutHelpFlags.CmdNewJob;
      A(;	//[5.0]
      AN    #Par.Status.AcceptNewSendData;
      A     #Par.OutHelpFlags.CmdNewJob;
      O;
      A     #Par.Status.WtTotalReached_InPos;
      A     #InRestdischarge;
      );	//[5.0]
      AN    #Par.ParMZDE;	//[5.0]
      S     #Par.Command.ResetWtTotal;
//==============================
      A     #InRestdischarge;
      AN    #Par.ParMZDE;	//[6.0]
      =     #Par.Command.OverwriteLL;
      A     #InRestdischarge;	//[6.0]
      A     #Par.ParMZDE;	//[6.0]
      =     #Par.Command.Restdischarge;	//[6.0]
//==============================
      A     #Par.Status.NewDataReady;
      =     #Par.Command.AcceptNewDataReady;
//==============================
      SET;
      =     #Par.Command.CommandReady;
//==============================
      A     #Par.Status.NewRcvData;
      =     #Par.Command.AcceptNewRcvData;
//==============================
      AN    #Par.Status.AcceptNewSendData;
      =     #Par.Command.NewSendData;
DP_B: NOP   0;
NETWORK
TITLE = (Profibus) Send Data
      A     #Par.ParOpto22;
      JC    DP_C;
//======================================================
//Test Send Dataset 000 done
      L     #DPData.NrSndDataSet;
      L     0;
      <>I;
      JC    s128;
      JU    S128;	//-->send 128
//------------------------------------------------
//Test Send Dataset 128 done
s128: L     #DPData.NrSndDataSet;
      L     128;
      <>I;
      JC    s136;
      AN    #Par.Status.WrongValue;
      A     #Par.OutHelpFlags.CmdNewValue;
      A     #CmdNewValue;
      R     #Par.OutHelpFlags.CmdNewValue;
      R     #CmdNewValue;
      JU    S136;	//-->Send 136
//------------------------------------------------
//Test Send Dataset 136 done
s136: L     #DPData.NrSndDataSet;
      L     136;
      <>I;
      JC    S000;
      JU    S128;	//-->Send 128
//==================================================
//Send Dataset 128
S128: A     #CmdNewValue;
      ON    #Par.Status.WtTotalReached_InPos;
      O     #InRestdischarge;
      JCN   S000;	//-->Send S000
      A     #CmdNewValue;
      =     #Par.OutHelpFlags.CmdNewValue;
      L     128;
      T     #DPData.NrSndDataSet;
      L     0;
      T     #DPData.IdxSndDataSet;
      AN    #Par.ParMZDE;	//[5.0]
      JC    S8DE;	//[5.0]
      L     #InFlowrate;	//[5.0]
      SLD   16;	//[5.0]
      T     #DPData.Data[1];	//[5.0]
      L     0;	//[5.0]
      T     #DPData.Data[2];	//[5.0]
      T     #DPData.Data[3];	//[5.0]
      T     #DPData.Data[4];	//[5.0]
      JU    send;	//[5.0]
S8DE: L     #InFlowrate;
      T     #DPData.Data[1];
      A     #InRestdischarge;
      L     0;
      JC    S8g1;
      L     #InJobWeight;
S8g1: T     #DPData.Data[2];
      L     0;
      T     #DPData.Data[3];
      L     #InRecipeNr;
      SLD   16;
      T     #DPData.Data[4];	//-->Byte 21
      JU    send;
//======================================================
//Send Dataset 136
S136: JU    S000;
      JU    send;
//======================================================
//Send Dataset 0
S000: L     0;
      T     #DPData.NrSndDataSet;
      L     0;
      T     #DPData.IdxSndDataSet;
send: CALL  "SIEMENS_BLKMOV" (
           SRCBLK                   := #Par.Command,
           RET_VAL                  := #tmpReturn,
           DSTBLK                   := #DPData.StatusCommand);
      A     #InSimulation;
      JC    sSim;
      CALL  "SIEMENS_DPWR_DAT" (
           LADDR                    := #tmpAddr,
           RECORD                   := #DPData,
           RET_VAL                  := #tmpReturn);
      L     #tmpReturn;
      L     0;
      <>I;
      =     #Par.OutHelpFlags.OutComFaultSend;
      JU    DP_C;
//write to Simulation
sSim: R     #Par.OutHelpFlags.OutComFaultSend;
      A     "GCS7_Gr_SimDPtoImage";
      L     P#Q 0.0;
      JC    rDB2;
      OPN   "TEST_IOSimuliOutput";
      L     P#DBX 0.0;
rDB2: L     #Par.ParIOByteNr;
      SLD   3;
      +D;
      LAR1;
      L     #DPData.StatusCommand;
      T     D [AR1,P#0.0];
      L     #DPData.NrSndDataSet;
      T     B [AR1,P#4.0];
      L     #DPData.IdxSndDataSet;
      T     B [AR1,P#5.0];
      L     #DPData.NrRcvDataSet;
      T     B [AR1,P#6.0];
      L     #DPData.IdxRcvDataSet;
      T     B [AR1,P#7.0];
      L     #DPData.Data[1];
      T     D [AR1,P#8.0];
      L     #DPData.Data[2];
      T     D [AR1,P#12.0];
      L     #DPData.Data[3];
      T     D [AR1,P#16.0];
      L     #DPData.Data[4];
      T     D [AR1,P#20.0];
DP_C: NOP   0;
NETWORK
TITLE = Automatical SetZeroPoint
      A     #Par.ParMZAH;
      O     #Par.ParMZDE;	//[5.0]
      JC    inZ1;	//[3.0]
      AN    "GCS7_Gr_OutTick1min";	//[3.0] Gr.OutTick1min;           
      JC    inZ0;	//[3.0]
      L     32000;	//[3.0]
      L     #OutSetZeroTime;	//[3.0]
      <I;	//[3.0]
      JC    inZ0;	//[3.0]
      +     1;	//[3.0]
      T     #OutSetZeroTime;	//[3.0]
inZ0: L     #OutSetZeroTime;	//[3.0]
      L     10000;	//[3.0]
      <I;	//[3.0]
      ON    #StStopped;	//[3.0]
      O     #tmpLocal;	//[3.0]
      JC    inZ1;	//[3.0]
      L     0;	//[3.0]
      T     #OutSetZeroTime;	//[3.0]
      S     #CmdSetZeroPoint;	//[3.0]
inZ1: NOP   0;
NETWORK
TITLE = States
//===State machine===
      A     #StStopped;
      JC    S0;
      A     #StStarting;
      JC    S1;
      A     #StStarted;
      JC    S2;
      A     #StStopping;
      JC    S3;
      A     #StFault;
      JC    S4;
      S     #StStopped;	//Init
      JU    S0;
NETWORK
TITLE =  StStopped
xxS0: S     #StStopped;
      R     #StStarted;
      JU    LOGX;
S0:   A     #tmpFault;
      R     #StStopped;
      JC    xxS4;	////--> Transition to StFault
      A     #Par.Status.Operation;
      AN    #OutComFault;	//[5.2]
      O;	//[2.1]
      AN    #OutStopPoint;	//[2.1]
      A     #Par.Command.Start;
      AN    #InRestdischarge;	//[2.3]
      R     #StStopped;
      JC    xxS1;	//--> Transition to StStarting
      JU    OUT;
NETWORK
TITLE =  StStarting
xxS1: S     #StStarting;
      R     #Par.OutHelpFlags.OutAlarmTimeOut;
      L     #Par.ParMonTime;
      T     #Par.OutMonTime;
      JU    OUT;
S1:   A     #tmpFault;	//Condition for StFault
      R     #StStarting;
      JC    xxS4;	//--> Transition to StFault
      A     #tmpOff;
      R     #StStarting;
      JC    xxS3;	//--> Transition to StStopping
      A     #Par.Status.Operation;
      R     #StStarting;
      JC    xxS2;	//--> Transition to StStarted
      JU    OUT;
NETWORK
TITLE =  StStarted
xxS2: S     #StStarted;
      JU    LOGX;
S2:   A     #tmpFault;	//Condition for StFault/StFalse
      R     #StStarted;
      JC    xxS4;	//--> Transition to StFault
      A     #tmpOff;
      ON    #Par.Status.Operation;
      R     #StStarted;
      JC    xxS3;	//--> Transition to StStopping
      JU    OUT;
NETWORK
TITLE =  StStopping
xxS3: S     #StStopping;
      R     #Par.OutHelpFlags.OutAlarmTimeOut;
      A     #OutSetZeroPoint;	//[3.0]
      JC    S3cc;	//[3.0]
      L     #Par.ParMonTime;
      T     #Par.OutMonTime;
S3cc: A     #StFault;
      R     #StFault;
      JC    LOGC;	//-->Message Operator ('fault cancelled' )
//State StStopping
S3:   A     #tmpFault;
      AN    #tmpLocal;
      R     #StStopping;
      JC    xxS4;	//-->Transition to StFault
//[7.3]      U     #tmpOn
//[7.3]      UN    #OutStopPoint               //[5.0]
//[7.3]      R     #StStopping
//[7.3]      SPB   xxS1                        //-->Transition to StStarting 
      L     2;	//[7.3] [7.6]
      L     #OutLCStep;	//[7.3]
      >=I;	//[7.3] [7.6]
      AN    #Par.Status.Operation;
      O     #OutComFault;	//[5.2]
      R     #StStopping;
      JC    xxS0;	//-->Transition to StStopped 
      JU    OUT;
NETWORK
TITLE =  FAULT
// State Fault
S4:   AN    #tmpFault;	//---Condition for StStopping
      A     #Par.OutHelpFlags.OutTestNewAlarm;
      O     #tmpLocalFault;
      JC    xxS3;	// Transition to StStopping
      A     #Par.OutHelpFlags.OutTestNewAlarm;
      JC    xxS4;
      JU    OUT;
NETWORK
TITLE = LOG
xxS4: S     "GCS7_Gr_InFaultFlag";	//Gr.InFaultFlag
      S     #StFault;
      R     #Par.OutHelpFlags.OutFaultResetDone;
      R     #Par.OutHelpFlags.OutTestNewAlarm;
      CALL  "SYS_Horn_Code" (
           FcCode                   := 1,
           ParObjectType            := 1028,
           ParObjectNo              := #Par.ParObjectNo,
           ParHornCode              := #Par.ParHornCode);
      L     #Par.ParMonTime;
      T     #Par.OutMonTime;
//Alarm Communication
      L     B#(1, 96);
      A     #OutComFault;
      JC    LOG;
//Tiemout
      A     #Par.OutHelpFlags.OutAlarmTimeOut;
      L     B#(1, 94);	// Message ('fault timeout')
      JC    LOG;
//Alarm-Nr 1..80
      L     0;
      L     #OutAlarmNr;
      ==I;
      JC    LOG2;
      L     B#(1, 0);
      OW;
      JU    LOG;	//Alarms 1..80
//Fault Remote Control
LOG2: L     B#(1, 90);	// Message ('fault DP Mode')   //[5.2]
      AN    #Par.Status.RemoteControl;	//[5.2]
      AN    #Par.ParOpto22;	//[5.2]
      JC    LOG;	//[5.2]
//Fault Wrong Value
      A     #Par.Status.WrongValue;
      L     B#(1, 95);	// Message ('fault wrong value')
      JC    LOG;
//Collected Alarm
      L     B#(1, 99);	// Message ('fault collected alarm')
      JU    LOG;
//===============================================
//State Transition
LOGX: AN    #tmpReport;
      JC    OUT;
      A     #StStopped;
      L     B#(4, 91);	//Message ('Stopped')
      JC    LOG;
      A     #StStarted;
      L     B#(4, 92);	//Message ('Dosing')
      JC    LOG;
      JU    OUT;
LOGC: L     B#(4, 0);	//Message ('fault cancelled')
LOG:  A     #Par.ParLogOff;	//---Set LOG Message
      JC    SAVE;
      T     #tmpLOGvalue;
      L     W#16#FF;
      AW;
      T     #OutAlarmNrLog;
      CALL  "GCS7_LogConvert" (
           ObjectNo                 := #Par.ParObjectNo,
           MsgType                  := #Par.ParMsgType,
           ClassMsgTxt              := #tmpLOGvalue,
           OType                    := 1026);	//LOG Message Converter / Entry / Contains Class and TextNo
SAVE: NOP   0;
NETWORK
TITLE = (Opto22) Communication start
//Prepare Telegram for send
OUT:  AN    #Par.ParOpto22;
      JC    OUT2;
      A     DBX 50.0;	//COM.LC0.CmdPut
      O     DBX 50.1;	//COM.LC0.CmdGet
      JC    OUT2;
//--- 'd'
      AN    #Par.OutComFlags.d_Done;
      AN    #Par.ParMZAH;
      AN    #Par.ParMZDE;	//[5.0]
      S     #Par.OutComFlags.d_Done;
      L     'd';
      JC    GET;
//--- 'i'
      AN    #Par.OutComFlags.i_Done;
      AN    #Par.ParMZAH;
      AN    #Par.ParMZDE;	//[5.0]
      S     #Par.OutComFlags.i_Done;
      L     'i';
      JC    GET;
      A     #Par.ParMZDE;	//[5.0]
      O     #Par.ParMZAH;
      AN    #Par.OutComFlags.h_done;
      S     #Par.OutComFlags.h_done;
      L     'h';
      JC    GET;
//--- 'P','Q'
      AN    #CmdNewValue;
      AN    #Par.OutHelpFlags.CmdNewValue;
      O     #Par.ParMZAH;
      O     #Par.ParMZDE;	//[5.0]
      JC    CmdK;
      A     #CmdNewValue;
      AN    #Par.OutHelpFlags.CmdNewValue;
      R     #CmdNewValue;
      S     #Par.OutHelpFlags.CmdNewValue;
      AN    #Par.OutComFlags.Q_Done;
      AN    #Par.ParWithFlowratePc;
      S     #Par.OutComFlags.Q_Done;
      L     'Q';
      JC    PUT;
      AN    #Par.OutComFlags.P_Done;
      A     #Par.ParWithFlowratePc;
      S     #Par.OutComFlags.P_Done;
      L     'P';
      JC    PUT;
//2A:--- 'K': not executed with zero setpoint or system adjust 
CmdK: AN    #CmdCorrFactor;
      AN    #Par.OutHelpFlags.CmdCorrFactor;
      O     #OutSetZeroPoint;
      O     #OutSystemAdjust;
      AN    #Par.ParMZDE;	//[5.0]
      JC    CmdS;
      A     #CmdCorrFactor;
      AN    #Par.OutHelpFlags.CmdCorrFactor;
      R     #CmdCorrFactor;
      S     #Par.OutHelpFlags.CmdCorrFactor;
      AN    #Par.OutComFlags.K_Done;
      AN    #Par.ParMZDE;	//[5.0]
      S     #Par.OutComFlags.K_Done;
      L     'K';
      JC    PUT;
//--- 'S'
CmdS: A     #Par.OutComFlags.S_Done;
      O     #Par.OutComFlags.A_Done;
      JC    CmCR;
      A     #Par.Status.Operation;
      X     #Par.Command.Start;	// ..if both signals are different
      O;
      A     #tmpFlag;
      AN    #Par.Command.Start;	// ..if both signals are different
      O     #CmdFaultReset;
      O     #CmdNewJob;
      O     #Par.OutHelpFlags.CmdNewValue;
      O     #CmdNewValue;
      O     #CmdSetZeroPoint;
      O     #Par.Command.ResetWtTotal;
      O     #Par.Command.ResetAlarm;
      JCN   CmCR;
      A     #Par.ParMZAH;
      O     #Par.ParMZDE;
      A     #CmdNewValue;
      AN    #Par.OutHelpFlags.CmdNewValue;
      R     #CmdNewValue;
      S     #Par.OutHelpFlags.CmdNewValue;
      A     #CmdNewJob;
      R     #CmdNewJob;
      S     #Par.Command.ResetWtTotal;
      A     #CmdFaultReset;
      R     #CmdFaultReset;
      S     #Par.Command.ResetAlarm;
      R     #Par.OutHelpFlags.OutAlarmTimeOut;
      A     #CmdSetZeroPoint;
      A     #StStopped;	//[3.0]
      R     #CmdSetZeroPoint;
      S     #Par.Command.SetZeroPoint;
      AN    #Par.ParMZAH;
      AN    #Par.ParMZDE;	//[5.0]
      S     #Par.OutComFlags.S_Done;
      L     'S';
      JC    PUT;
      S     #Par.OutComFlags.A_Done;
      L     'A';
PUT:  SET;
      S     DBX 50.0;	//COM.LC0.CmdPut ;
      JU    ALL1;
GET:  SET;
      S     DBX 50.1;	//COM.LC0.CmdGet ;
ALL1: T     DBB 51;	//COM.LC0.Command;
      JU    OUT2;
// 
//---Clear command flags (x_done)
CmCR: R     #Par.OutComFlags.i_Done;
      R     #Par.OutComFlags.d_Done;
      R     #Par.OutComFlags.h_done;
      R     #Par.OutComFlags.Q_Done;
      R     #Par.OutComFlags.P_Done;
      R     #Par.OutComFlags.S_Done;
      R     #Par.OutComFlags.K_Done;
      R     #Par.OutComFlags.A_Done;
NETWORK
TITLE = Global End
OUT2: A     #StStarted;
      O     #StStarting;
      AN    #tmpOff;
      AN    #tmpLocal;
      =     #OutpDosingEnable;
      SET;	//---Clear all commands
      R     #CmdOff;
      R     #CmdOn;
      R     #CmdNext;
//--Output for group 
      AN    #InLocal;
      O     #InManual;
      A     #InDPFault;
      S     "GCS7_Gr_InDPFault";
      AN    #InLocal;
      O     #InManual;
      A     #InHWStop;
      S     "GCS7_Gr_InHWStop";
NETWORK
TITLE = State Code
//--Stopped, Substate ---
      AN    #StStopped;
      JC    STC2;
      L     41;	//Code: StStopped.HWStop
      A     #InHWStop;
      JC    STC;
      L     51;	//Code: StStopped.DPFault
      A     #InDPFault;
      JC    STC;
      L     1;	// Code: stopped
      JC    STC;
//--------------------
STC2: L     2;	//Code: StStarting
      A     #StStarting;
      JC    STC;
      L     3;	//Code: StStarted
      A     #StStarted;
      JC    STC;
      L     7;	//Code: StStopping
      A     #StStopping;
      JC    STC;
      L     32;	//Code: fault
STC:  L     #StCode;	//Old state code
      TAK;
      T     #StCode;	//Save state code
      <>I;
      L     3;	//Load code for CBit methode
      CC    "SYS_CBitCtrl";
NETWORK
TITLE =  Store LC data
      AN    #Par.ParOpto22;
      BEC;
      L     #Par.ParLCIdx;
      T     DBW 34;	//COM.Element.Index; 
      L     2;	//Store LC data
      T     DBW 0;	//COM.CODE;
      CDB;
      UC    "GCS7_RS485Ctrl";
      CDB;
STOR: BEU;
END_FUNCTION_BLOCK

FUNCTION_BLOCK "GCS7_E_Sampler"	// FB 29
TITLE = Sampler MZER + MZEP
// 
//COPYRIGHT:    (C) 1997  BUHLER AG, CH-9240 UZWIL, SWITZERLAND
//
//PRODUCT:      GCS7
//
//TITLE:        Element Sampler MZER + MZEP
//              (GCPROVB Revision=12)
//-------------------------------------------------------------------------
//
//IDENT:        AUTHOR:             DEPT:                       DATE:
//FB29.7.2      A. Egli             CT3                         13-Sep-2007
//              Send InSimulation to tag reader
//FB29.7.1      A. Egli             CT3                         30-Mai-2007
//              ProfibusDP: Line LAR1 moved
//FB29.7.0      A. Egli             CT3                         14-Mar-2007
//              - Using Baumer FB to read RFID
//              - OutBottleInPosition
//              - InSimulation  
//              - Do not read IO as long DPNode is not connected
//              - CmdFaultReset: Reset OutNxBottleNotEmpty, OutCoverNotClosed 
//FB29.6.2      Ph. Engler          GP92                        21-Feb-2007
//              - Changes for failure save tag reading
//              - Changes for Tag registration
//FB29.6.1      A. Egli             CT3                         19-Jun-2006
//              Reading Tag only when bottle in position
//FB29.6.0      Ph. Engler          MU92                        14-Feb-2006
//              - Tag reading corrected
//FB29.5.2      Ph. Engler          MU92                        01-Sep-2005
//              - Don't reset Sample and BottleChangeTime if no productflow
//              - Reload InBottleChangeTime on every StBottleChange
//FB29.5.1      A. Egli             CT3                         17-Mai-2005
//              CmdBottleChange do not delete OutSampleCounter
//              (only when ParBatchSampler=1)
//FB29.5.0      A. Egli             CT3                         05-Mai-2004
//              2kByte or 256 Byte
//FB29.4.2      A. Egli             CT3                         24-Sep-2003
//              Alarm handling 
//FB29.4.1      A. Egli             CT3                         04-Sep-2003
//              Write outputs only to peripherie not to image
//FB29.4.0      A. Egli             CT3                         10-Mai-2003
//              New Release with one block , Profibus-DP, Tag-Reader
//FB29.3.0      S. Kalberer         CT3                         21-Feb-2000
//              MZEP added, new reLOG 17
//FB29.2A       A. Egli             CT3                         04-Mai-1998
//              StFault = StCode 32
//FB29.1A       S. Kalberer         AEE61                       31-Jul-1997
//              1st Release in S7
//
//-------------------------------------------------------------------------
//
//PURPOSE:      MANUAL : see [MZExxMAN]
//
//RESTRICTIONS: S7
//              ACCU2: Pointer to dynamic datas of the element
//              ACCU1: Pointer to parameter datas of the element
//
//-------------------------------------------------------------------------
//=======================================================
//Log Message: 
//------------------------------------------------------
// 0   off
// 1   wait
// 2   sampling
// 3   bottle change
// 4   sampler in local mode
// 9   fault cancelled
//10  fault sampling
//11  fault sample time
//12  fault current bottle full
//13  fault bottle change (reLOG fault)
//14  fault next bottle not empty
//15  fault cover not closed
//16  fault multiple
//18  fault reading RFID
//=======================================================
//StCode:  State               
//------------------------------------------------------
//32       StFault                 
// 1       StOff                   
//41       StOff.HWStop                     StOff + InHWStop
//51       StOff.DPFault                    StOff + InDPFault
// 2       StWait                
// 3       StSampling              
// 4       StBottleChange        
// 5       StWarning             
//45       StWarning.HWStop                 StWarning + InHWStop
//55       StWarning.DPFault                StWarning + InDPFault
//
//
AUTHOR : EA
FAMILY : GCS7LL
NAME : MZEx
VERSION : 7.2
VAR
  StCode : INT ;	//Element state code
  InEnable : BOOL ;	//Interlocking: 1= Enable to start/ 0= Immediate stop
  spare0201 : BOOL ;
  InSimulation : BOOL ;
  OutReadingFaultRFID : BOOL ;	//Reading Fault RFID
  CmdSendResult : BOOL ;
  InpSampleAllowed : BOOL ;	//DI sample allowed (2*)
  InpBottleChangeAllowed : BOOL ;	//DI botte change allowed (2*)
  InProductFlow : BOOL ;	//Signal to indicate product flow in automatic mode
  CmdSample : BOOL ;	//Pulse to start a sample sequence
  CmdBottleChange : BOOL ;	//Pulse to start a bottle change sequence
  CmdNewBatch : BOOL ;	//Pulse to start a new batch (for batch sampler only)
  CmdFaultReset : BOOL ;	//Command to reset fault
  InLocal : BOOL ;	//1= Local mode (no fault by start with service switch)
  InManual : BOOL ;	//1= Manual/ 0= Automatic
  InReport : BOOL ;	//Report of all state transitions
  InWarningMode : BOOL ;	//1= By fault, the element changes to StWarning
  InHWStop : BOOL ;	//HW stop is detected, no fault
  InDPFault : BOOL ;	//DP-Fault is detected, no fault
  OutProductFlow : BOOL ;	//Signal product flow
  OutDelayFault : BOOL ;	//Signal delay time over
  OutFlagOk : BOOL ;	//Signal positive edge flag ok (2*)
  OutBottleInPosition : BOOL ;
  OutResponseFault : BOOL ;	//Signal response time over
  OutResponseTime : BOOL ;	//Signal response time running
  StOff : BOOL ;	//Element is off
  StWait : BOOL ;	//Element is on and waiting for next steps
  StSampling : BOOL ;	//Element is sampling
  StBottleChange : BOOL ;	//Element is changing bottle
  StFault : BOOL ;	//Element has a fault
  StWarning : BOOL ;	//Element has a warning
  spare56 : BOOL ;
  spare57 : BOOL ;	//
  InpSamplerInAuto : BOOL ;	//DI sampler in automatic mode (1*/2*)
  InpCmdOk : BOOL ;	//DI command ok (1*)
  InpAlarmCollect : BOOL ;	//DI alarm collected (1*)
  InpAlarmSampleTime : BOOL ;	//DI alarm sample time (1*)
  InpAlarmCurBottleFull : BOOL ;	//DI alarm current bottle full (1*)
  InpAlarmNxBottleNotEmpty : BOOL ;	//DI alarm next bottle not empty  (1*/2*)
  InpAlarmCoverNotClosed : BOOL ;	//DI alarm cover not closed  (1*)
  InpAlarmMultiple : BOOL ;	//DI alarm multiple (for further alarms)  (1*)
  OutCurBottleFull : BOOL ;	//Signal current bottle full
  OutNxBottleNotEmpty : BOOL ;	//Signal next bottle not empty
  OutCoverNotClosed : BOOL ;	//Signal cover not closed
  OutSamplerInLocal : BOOL ;	//Signal sampler in local mode
  OutpAlarmReset : BOOL ;	//DO alarm reset  (1*)
  OutpSampling : BOOL ;	//DO sampling (1*/2*)
  OutpBottleChange : BOOL ;	//DO change bottle (1*/2*)
  OutpFuncRelease : BOOL ;	//DO function release (1*)
  InSamplePerBatch : INT ;	//Number of sample per batch
  InSampleTime : INT ;	//Time between two samples [s]
  InBottleChangeTime : INT ;	//Time between two bottle changes [s]
  OutSampleCounter : INT ;	//Actual value: Sample counter
  OutBottleCounter : INT  := 1;	//Actual value: Bottle counter
  OutActSampleTime : INT ;	//Actual time: Before next sample [s]
  OutActBottleChangeTime : INT ;	//Actual time: Before next bottle change [s]
  InSamplePulseLength : INT ;	//Lenght of Sample pulse lenght [ms]
  Tag : STRUCT
   HskWrite : STRUCT
    Q_Result : BOOL ;
   END_STRUCT ;
   HskRead : STRUCT
    F_Result : BOOL ;
   END_STRUCT ;
   OutRegistrated : BOOL ;
   InJobNr : DINT ;	//Current Job
   InBatchNr : INT ;	//Current batch
   OutTagNrAc : DWORD ;	//Tag number of the current bottle
   OutJobNrResult : DWORD ;	//Job number of the resulting bottle
   OutBatchNrResult : INT ;	//Batch number of the resulting bottle
   OutTagNrResult : DWORD ;	//Tag number of the resulting bottle
   spare_1 : DWORD ;
   spare_2 : DWORD ;
  END_STRUCT ;
  OutAlarmNrLog : INT ;	//Last textnumber send to log
  Par : STRUCT
   ParObjectNo : INT ;	//Is used for communication with PC, e.g. for message
   ParMsgType : INT ;	//Is used for message (translation of state)
   ParHornCode : INT ;	//Is used by horn module
   ParLogOff : BOOL ;	//Report is off
   spare0401 : BOOL ;
   ParBatchSampler : BOOL ;	//1= Batch sampler / 0= Job sampler
   ParBatchBottleChange : BOOL ;	//1= Automatic bottle change with batch sampler
   ParMZEP : BOOL ;	//1= Sampler MZEP / 0= Sampler MZER
   ParAlarmCollectWarn : BOOL ;	//InpAlarmCollect gives only warning
   ParAlarmSampleTimeWarn : BOOL ;	//InpAlarmSampleTime gives only warning
   ParAlarmCurBottleWarn : BOOL ;	//InpAlarmCurBottleFull gives only warning
   ParAlarmNxBottleWarn : BOOL ;	//InpAlarmNxBottleNotEmpty gives only warning
   ParAlarmCoverWarn : BOOL ;	//InpAlarmCoverNotClosed gives only warning
   ParAlarmMultipleWarn : BOOL ;	//InpAlarmMultiple gives only warning
   ParDP : BOOL ;	//Profibus DP
   ParTagReader : BOOL ;	//OIS Tagreader
   ParIOByteNr : INT ;	//PROFIBUS: Address of first input and output byte Profibus DP
   ParDBNoRFID : INT ;	//Instance DB of SSA_EL_Sampler_RFID
   ParSampleResponseTime : INT ;	//Maximum response time after CmdSample
   ParBottleResponseTime : INT ;	//Maximum response time after CmdBottleChange
   ParAlarmResponseTime : INT ;	//Maximum response time after CmdFaultReset
   ParDelayTime : INT ;	//Delay time after InProductFlow
   OutActResponseTime : INT ;	//Actual time: Response time
   OutActDelayTime : INT ;	//Actual time: Delay time after InProductFlow
   OutSpare22 : INT ;
   OutSpare26 : INT ;
   OutSpare28 : DINT ;
  END_STRUCT ;
END_VAR
VAR_TEMP
  tmpLOGvalue : WORD ;	//LOG value
  tmpLenDyn : DINT ;
  tmpReport : BOOL ;	//Global LOG all
  tmpFaultReset : BOOL ;	//Global FaultReset
  tmpWarning : BOOL ;	//temp sampler warning
  tmpFault : BOOL ;	//temp sampler fault
  tmpResponseFault : BOOL ;	//temp sampler response fault
  tmpAlarmCollect : BOOL ;	//temp sampler alarm collect
  tmpEnableWait : BOOL ;	//Enable to change to StWait (automatic mode)
  tmpEnableManual : BOOL ;	//Enable manual mode
  tmpCmdOk : BOOL ;	//temp sampling/bottle change is finished and ok
  tmpLocal : BOOL ;
  tmpLocalFault : BOOL ;
  InpData : STRUCT
   KDO : BYTE ;
   ANT : BYTE ;
   StartP : BYTE ;
   AnzP : BYTE ;
   ADB : BYTE ;
   DBN : BYTE ;
   DBL : BYTE ;
   CTR : BYTE ;
  END_STRUCT ;
  OutpData : STRUCT
   KDO : BYTE ;
   ANT : BYTE ;
   StartP : BYTE ;
   AnzP : BYTE ;
   ADB : BYTE ;
   DBN : BYTE ;
   DBL : BYTE ;
   CTR : BYTE ;
  END_STRUCT ;
  tmpAddrIO : DWORD ;
  tmpIO : STRUCT
   AE32_0 : BOOL ;
   AE32_1 : BOOL ;
   AE32_2 : BOOL ;
   AE32_3 : BOOL ;
   AE32_4 : BOOL ;
   AE32_5 : BOOL ;
   AE32_6 : BOOL ;
   AE32_7 : BOOL ;
   AE33_0 : BOOL ;
   AE33_1 : BOOL ;
   AE33_2 : BOOL ;
   AE33_3 : BOOL ;
   AE33_4 : BOOL ;
   AE33_5 : BOOL ;
   AE33_6 : BOOL ;
   AE33_7 : BOOL ;
   EAW102 : INT ;
  END_STRUCT ;
  tmpAddrDP : DWORD ;
  tmpSendResult : BOOL ;
  tmpDBTagReader : INT ;
END_VAR
BEGIN
NETWORK
TITLE =  Start Global
      L     92;
      T     #tmpLenDyn;	//--> Len dynamic data in byte
NETWORK
TITLE = PC Control
//=== Test Object number =====================
      L     "SYS_DirectCtrlDB".PC.ObjectNo;	//PCControl.ObjectNo
      L     #Par.ParObjectNo;	//Input ObjectNo
      <>I;
      JC    Ctrl;
//=== Test OType      ========================
      L     1029;	//Input object type
      L     "SYS_DirectCtrlDB".PC.ObjectType;	//PCControl.ObjectType
      <>I;
      JC    Ctrl;
//=== Test Handshake =========================
      A     "SYS_DirectCtrlDB".PC.Hsk.FExamine;	//Handshake.FExamine
      JC    pExa;
      A     "SYS_DirectCtrlDB".PC.Hsk.FDefineCmd;	//Handshake.FDefineCmd
      JC    pCmd;
      A     "SYS_DirectCtrlDB".PC.Hsk.FDefinePara;	//Handshake.FDefinePara
      JC    pPar;
pIni: L     2;	//FcInit
      UC    "SYS_DirectCtrl";
      JU    Ctrl;
//Write parameter 
pPar: LAR1  P#DBX 58.0;
      L     P##Par;
      L     DW#16#FFFFF;
      AD;
      +AR1;
      L     DBW [AR1,P#8.0];
      T     #Par.ParSampleResponseTime;
      L     DBW [AR1,P#10.0];
      T     #Par.ParBottleResponseTime;
      L     DBW [AR1,P#12.0];
      T     #Par.ParAlarmResponseTime;
      L     DBW [AR1,P#14.0];
      T     #Par.ParDelayTime;
//Write new commands from PC to Interface of group 
pCmd: A     "SYS_DirectCtrlDB".PC.Cmd1[0];	//Cmd1[0]  =Q_Result
      S     #Tag.HskWrite.Q_Result;
      A     "SYS_DirectCtrlDB".PC.Cmd1[8];	//Cmd1[8]  =CmdSample
      S     #CmdSample;
      A     "SYS_DirectCtrlDB".PC.Cmd1[9];	//Cmd1[9]  =CmdBottleChange
      S     #CmdBottleChange;
      A     "SYS_DirectCtrlDB".PC.Cmd1[10];	//3.0: Cmd1[10] =CmdNewBatch
      S     #CmdNewBatch;
      A     "SYS_DirectCtrlDB".PC.Cmd1[11];	//Cmd1[11] =CmdFaultReset
      S     #CmdFaultReset;
      A     "SYS_DirectCtrlDB".PC.Cmd1[13];	//Cmd1[13]=CmdManualOn
      S     #InManual;
      A     "SYS_DirectCtrlDB".PC.Cmd2[13];	//Cmd2[13]=CmdManualOff
      R     #InManual;
      A     "SYS_DirectCtrlDB".PC.Cmd1[14];	//Cmd1[14]=CmdReportOn
      S     #InReport;
      A     "SYS_DirectCtrlDB".PC.Cmd2[14];	//Cmd2[14]=CmdReportOff
      R     #InReport;
      A     "SYS_DirectCtrlDB".PC.Cmd1[15];	//Cmd1[15]=CmdWarningOn
      S     #InWarningMode;
      A     "SYS_DirectCtrlDB".PC.Cmd2[15];	//Cmd2[15]=CmdWarningOff
      R     #InWarningMode;
//Define Value
      AN    "SYS_DirectCtrlDB".PC.Hsk.FDefineValue;	// PC.Hsk.FDefineValue
      ON    #InManual;
      JC    pIni;
      LAR1  P#DBX 58.0;
      L     DBD [AR1,P#8.0];
      T     #InSamplePerBatch;
      L     DBD [AR1,P#10.0];
      T     #InSampleTime;
      L     DBW [AR1,P#12.0];
      T     #InBottleChangeTime;
      JU    pIni;
pExa: TAR2;	//Address dynamic datas
      T     "SYS_DirectCtrlDB".GC.InDynAddr;	//-->PCControl.GC.InDynAddr
      L     #tmpLenDyn;	//Length dynamic datas
      T     "SYS_DirectCtrlDB".GC.InDynLen;	//-->PCControl.GC.InDynLen
      L     0;
      T     "SYS_DirectCtrlDB".GC.InParaAddr;	//-->PCControl.GC.InParaAddr
      T     "SYS_DirectCtrlDB".GC.InParaLen;	//-->PCControl.GC.InParaLen
      L     1;	//Code FcExamine
      UC    "SYS_DirectCtrl";
      L     11;	//Revision   [5.0]
      T     "SYS_DirectCtrlDB".GC.Revision;
Ctrl: NOP   0;
NETWORK
TITLE = Read Data from Profibus DP
      AN    #Par.ParDP;
      JC    rdJ0;
      L     #Par.ParIOByteNr;
      SLD   3;
      T     #tmpAddrDP;
      LAR1;	//[7.1]
      L     0;	//[7.0]
      A     #InDPFault;	//[7.0]
      JC    rdJ2;	//[7.0]
      AN    #InSimulation;	//[7.0]
      JC    rdJ1;	//[7.0]
      L     ID [AR1,P#0.0];	//[7.0]
      JU    rdJ2;	//[7.0]
rdJ1: L     PID [AR1,P#0.0];
rdJ2: LAR1  P##tmpIO;
      T     LD [AR1,P#0.0];
      A     #tmpIO.AE33_0;
      =     #InpSamplerInAuto;
      A     #tmpIO.AE33_1;
      =     #InpCmdOk;
      A     #tmpIO.AE33_2;
      =     #InpAlarmCollect;
      A     #tmpIO.AE33_3;
      =     #InpAlarmSampleTime;
      A     #tmpIO.AE33_4;
      =     #InpAlarmCurBottleFull;
      A     #tmpIO.AE33_5;
      =     #InpAlarmNxBottleNotEmpty;
      A     #tmpIO.AE33_6;
      =     #InpAlarmCoverNotClosed;
      A     #tmpIO.AE33_7;
      =     #InpAlarmMultiple;
      L     2#100000000000000;	//[7.0] E32.6
      L     #tmpIO.EAW102;	//[7.0]
      AW;	//[7.0]
      ==I;	//[7.0]
      =     #OutBottleInPosition;	//[7.0]
rdJ0: NOP   0;
NETWORK
TITLE =  All State Init
//===Clear tmp Variable
//===Global Group Orders===
//---Report is on---
      A     "GCS7_Gr_OutReportAll";	//Gr.OutReportAll
      O     #InReport;
      =     #tmpReport;
//---FaultReset is on---
      A     "GCS7_Gr_OutFaultReset";	//Gr.OutFaultReset
      S     #CmdFaultReset;
      A     #CmdFaultReset;
      =     #tmpFaultReset;
//3.0:---Command Ok: dyn.InpCmdOk replaced with tmpCmdOk
      A     #Par.ParMZEP;
      A     #InpSampleAllowed;
      FP    #OutFlagOk;
      O;
      AN    #Par.ParMZEP;
      A     #InpCmdOk;
      =     #tmpCmdOk;
//---Manual mode---
      A     "GCS7_Gr_OutManualOff";	//Gr.OutManualOff
      R     #InManual;
      A     #InManual;
      S     "GCS7_Gr_InManual";	//Gr.InManual
//tmpLocal
      A     #InLocal;
      AN    #InManual;
      =     #tmpLocalFault;
      A     #tmpLocalFault;
      O     #InDPFault;
      O     #InHWStop;
      =     #tmpLocal;
//---tmpEnableWait: aux. signal to stay in state StWait
      A     #InEnable;	//Automatic
      AN    #InLocal;
      AN    #InManual;
      A     #OutpFuncRelease;
      AN    #tmpLocal;
      =     #tmpEnableWait;
//---tmpEnableManual: changing from StOff directly to StSampl./BottleChange
//   without 'InEnable' Interlocking
      A     #CmdSample;
      O     #CmdBottleChange;
      A     #InManual;
      A     #OutpFuncRelease;
      AN    #tmpLocal;
      =     #tmpEnableManual;
//===New batch
      AN    #CmdNewBatch;
      JC    inJ1;	//At CmdNewBatch
      L     0;	// do Clear sample counter
      T     #OutSampleCounter;
//===Warning/Fault detection
inJ1: AN    #InpAlarmCollect;	//[4.2]
      AN    #InpAlarmSampleTime;	//[4.2]
      AN    #InpAlarmCurBottleFull;	//[4.2]
      AN    #InpAlarmNxBottleNotEmpty;	//[4.2]
      AN    #InpAlarmCoverNotClosed;	//[4.2]
      AN    #InpAlarmMultiple;	//[4.2]
      AN    #OutReadingFaultRFID;	//[7.0]
      R     #tmpWarning;	//No warning, no fault
      R     #tmpFault;
      JC    FNC;
//---Save alarm info: Set Output OutXxx
      A     #InpAlarmCurBottleFull;
      S     #OutCurBottleFull;
      A     #InpAlarmNxBottleNotEmpty;
      S     #OutNxBottleNotEmpty;
      A     #InpAlarmCoverNotClosed;
      S     #OutCoverNotClosed;
      A     #OutpAlarmReset;	//[7.0]
      AN    #InpAlarmNxBottleNotEmpty;	//[7.0]
      R     #OutNxBottleNotEmpty;	//[7.0]
      A     #OutpAlarmReset;	//[7.0]
      AN    #InpAlarmCoverNotClosed;	//[7.0]
      R     #OutCoverNotClosed;	//[7.0]
//---Check for releavant Alarms
      A     #InpAlarmCollect;	//[4.2]
      AN    #Par.ParAlarmCollectWarn;	//[4.2]
      O;	//[4.2]
      A     #InpAlarmSampleTime;	//[4.2]
      AN    #Par.ParAlarmSampleTimeWarn;	//[4.2]
      O;	//[4.2]
      A     #InpAlarmCurBottleFull;	//[4.2]
      AN    #Par.ParAlarmCurBottleWarn;	//[4.2]
      O;	//[4.2]
      A     #InpAlarmNxBottleNotEmpty;	//[4.2]
      AN    #Par.ParAlarmNxBottleWarn;	//[4.2]
      O;	//[4.2]
      A     #InpAlarmCoverNotClosed;	//[4.2]
      AN    #Par.ParAlarmCoverWarn;	//[4.2]
      O;	//[4.2]
      A     #InpAlarmMultiple;	//[4.2]
      AN    #Par.ParAlarmMultipleWarn;	//[4.2]
      O;	//[7.0]
      A     #OutReadingFaultRFID;	//[7.0]
      A     #Par.ParTagReader;	//[7.0]
      =     #tmpFault;	//-->Fault detected
      AN    #tmpFault;	// Fault detected
      =     #tmpWarning;	//-->Warning detected
      A     #CmdBottleChange;	//[4.2]
      A     #InpAlarmCurBottleFull;	//[4.2]
      A     #tmpWarning;	//[4.2]
      S     #CmdFaultReset;	//[4.2]
FNC:  NOP   0;
NETWORK
TITLE =  Batch and Job sample functions
// !! Only in automatic mode !!
//
//=>Batch Sampler(ParBatchSampler='1', ParBatchBottleChange='0'):
//  The sampler takes several configured samples per batch into one 
//  bottle, without automatically changing the bottle.
//  If product flows (InProduct='1') it will take samples every InSampleTime
//  up to number of sample per batch (InSamplePerBatch).
//  With CmdNewBatch you can start a new sample sequence into the same bottle.
//  If it's necessary to change first the bottle and then start a new sample
//  sequence, use only CmdBottleChange (e.g. mixing lines).
//
//  With ParBatchBottleChange='1': It takes several configured samples per batch
//  into one bottle and changes automatically the bottle after InBottleChangeTime.
//
//=>Job Sampler (ParBatchSampler='0'):
//  The sampler takes samples and changes automatically the bottles
//  in configured time intervals.
//  If product flows (InProduct='1') it will take samples every
//  InSampleTime and changes the bottles every InBottleChangeTime
//  (e.g. blending lines or intake).
      AN    #tmpEnableWait;
      ON    "GCS7_Gr_OutTick1s";	//Gr.OutTick1S
      O     #StFault;
      O     #StWarning;
      JC    STAT;
//===Job or batch sampler active only in automatic mode
      AN    #Par.ParBatchSampler;
      JC    FNC1;
//---Samples per Batch reached: only Batch sampler
      L     #OutSampleCounter;
      L     #InSamplePerBatch;
      >=I;
      JC    FNC2;	//Batch finished: no sampling anymore
//----Sample intervall: Job and Batch Sampler
FNC1: L     #InSampleTime;	//Check InSampleTime >=0
      L     0;
      <=I;
      ON    #OutDelayFault;	//Delay time not over
      JC    FNC2;
      L     #OutActSampleTime;
      +     -1;
      T     #OutActSampleTime;
      <I;
      JC    FNC2;
      S     #CmdSample;	//Sampling time over, take now a sample
      L     #InSampleTime;	//set new time
      T     #OutActSampleTime;
//---Bottle change interval: Job or Batch Sampler with bottle change
FNC2: L     #InBottleChangeTime;	//Check InBottleChangeTime >=0
      L     0;
      <=I;
      ON    #OutDelayFault;	//Delay time not over
      O(;
      A     #Par.ParBatchSampler;	//Batch sampler without..
      AN    #Par.ParBatchBottleChange;	//..automatically bottle change
      );
      JC    FNC5;
      L     #OutActBottleChangeTime;
      +     -1;
      T     #OutActBottleChangeTime;
      <I;
      JC    FNC5;
      S     #CmdBottleChange;	//BottleChange time time over, change bottle now
      L     #InBottleChangeTime;	//set new time
      T     #OutActBottleChangeTime;
//---Delay sampling and bottle change with DelayTime
FNC5: A     #OutProductFlow;
      ON    #InProductFlow;
      JC    FNC6;
      S     #OutProductFlow;
      L     #Par.ParDelayTime;
      T     #Par.OutActDelayTime;
//[5.2]      L     #InSampleTime
//[5.2]      T     #OutActSampleTime
//[5.2]      L     #InBottleChangeTime
//[5.2]      T     #OutActBottleChangeTime
FNC6: AN    #OutProductFlow;
      O     #OutDelayFault;
      JC    STAT;
      L     #Par.OutActDelayTime;
      +     -10;
      T     #Par.OutActDelayTime;
      L     0;
      <=I;
      S     #OutDelayFault;	//DelayTime over
NETWORK
TITLE =  States
//===State machine===
STAT: A     #StOff;
      JC    S0;
      A     #StWait;
      JC    S1;
      A     #StSampling;
      JC    S2;
      A     #StBottleChange;
      JC    S3;
      A     #StFault;
      O     #StWarning;
      JC    S4;
      S     #StOff;	//Init
      JU    S0;
NETWORK
TITLE = StOff
//Any transition to StOff
xS0:  S     #StOff;
      R     #StWait;
      L     0;	//Reset actual timer
      T     #Par.OutActResponseTime;
      T     #Par.OutActDelayTime;
      AN    #InReport;
      JC    OUT;
      L     B#(4, 0);	//Message Info ('off' )
      JU    LOG;
//=== Logic ====
S0:   A     #tmpEnableWait;	//Condition for StWait
      O     #tmpEnableManual;
      JC    xS1;
      JU    OUT;
NETWORK
TITLE =  StWait
//Any Transition to StWait
xS1:  R     #StOff;
      AN    #tmpEnableManual;
      O     #tmpEnableWait;
      O     #tmpCmdOk;	//Old command is not finished yet
      JC    xS1a;
//Manual mode with no Interlocking
      A     #CmdSample;	//Condition for StSampling
      JC    xS2;
      JU    xS3;	//Condition for StBottleChange
//Automatic mode
xS1a: S     #StWait;
//Increment BottleCounter (ring counter 1-27)
      AN    #StBottleChange;
      JC    xS1s;
      R     #OutCurBottleFull;
      L     27;
      L     #OutBottleCounter;
      +     1;
      >=I;
      JC    xS1b;
      L     1;
xS1b: T     #OutBottleCounter;
      A     #Par.ParBatchSampler;	//[5.1]
      JC    xS1c;	//[5.1]
      L     0;	//Reset SampleCounter
      T     #OutSampleCounter;
xS1c: NOP   0;	//[5.1]
      AN    #Par.ParBatchSampler;
      JC    xS1r;	//At Batch sampler
      L     #InSampleTime;	// do Actualize sample time
      T     #OutActSampleTime;
      JU    xS1r;
//Increment Sample Counter
xS1s: AN    #StSampling;
      JC    xS1r;
      L     #OutSampleCounter;
      +     1;
      T     #OutSampleCounter;
xS1r: R     #StSampling;
      R     #StBottleChange;
      AN    #tmpEnableWait;	//Condition for immediate change to StOff
      JC    xS0;
      AN    #tmpReport;
      JC    OUT;
      L     B#(4, 1);	//Message Info ('wait')
      JU    LOG;
//=== Logic ====
S1:   AN    #tmpEnableWait;	//Condition for StOff
      JC    xS0;
      AN    #CmdNewBatch;
      JC    S1J1;	//At CmdNewBatch
      L     #InSampleTime;	// do Actualize sample time
      T     #OutActSampleTime;
S1J1: A     #InpSampleAllowed;	// 3.0:
      A     #Par.ParMZEP;	// 3.0:
      ON    #Par.ParMZEP;	// 3.0:
      A     #CmdSample;
      AN    #tmpCmdOk;
      JC    xS2;
      A     #InpBottleChangeAllowed;	// 3.0:
      A     #Par.ParMZEP;	// 3.0:
      ON    #Par.ParMZEP;	// 3.0:
      A     #CmdBottleChange;
      AN    #tmpCmdOk;
      JC    xS3;
      JU    OUT;	//Condition for StWait
NETWORK
TITLE = StSampling
//Any transition to StSampling
xS2:  S     #StSampling;
      R     #StWait;
      R     #CmdSample;
      L     #Par.ParSampleResponseTime;	//Set timer
      T     #Par.OutActResponseTime;
      AN    #tmpReport;
      JC    OUT;
      L     B#(4, 2);	//Message Info ('sampling')
      JU    LOG;
//=== Logic ====
//Transition to StWait
S2:   A     #tmpCmdOk;	//Condition for StWait
      JC    xS1;
      AN    "GCS7_Gr_OutTick1s";	//Gr.OutTick1S
      L     #Par.OutActResponseTime;
      JC    S2J1;
      +     -10;
      T     #Par.OutActResponseTime;
S2J1: L     0;
      <=I;
      S     #OutResponseFault;
      AN    #OutResponseFault;	//Condition for StSampling
      AN    #tmpFault;
      AN    #tmpWarning;
      JC    OUT;
      JU    xS45;	//Transition to StFault/StWarning
NETWORK
TITLE = StBottleChange
//Any transition to StBottleChange
xS3:  S     #StBottleChange;
      R     #StWait;
      R     #CmdBottleChange;
      R     #OutNxBottleNotEmpty;
      R     #OutCoverNotClosed;
      L     #Par.ParBottleResponseTime;	//Set timer
      T     #Par.OutActResponseTime;
      L     #InBottleChangeTime;	//[5.2]
      T     #OutActBottleChangeTime;	//[5.2]
      SET;
      S     #CmdSendResult;
      AN    #tmpReport;
      JC    OUT;
      L     B#(4, 3);	//Message Info ('bottle change')
      JU    LOG;
//=== Logic ====
//Transition to StWait
S3:   A     #tmpCmdOk;	//Condition for StWait
      JC    xS1;
      AN    "GCS7_Gr_OutTick1s";	//Gr.OutTick1S
      L     #Par.OutActResponseTime;
      JC    S3J1;
      +     -10;
      T     #Par.OutActResponseTime;
S3J1: L     0;
      <=I;
      S     #OutResponseFault;
      AN    #OutResponseFault;	//Condition for StBottleChange
      AN    #tmpFault;
      AN    #tmpWarning;
      JC    OUT;
      JU    xS45;	//Transition to StFault/StWarning
NETWORK
TITLE =  Fault/Warning
//Any transiton to Fault/Warning
xS45: A     #InpAlarmSampleTime;
      L     B#(1, 11);	//Message Error ('fault sample time')
      JC    S45a;
      A     #InpAlarmCurBottleFull;
      L     B#(1, 12);	//Message Error ('fault actual bottle full')
      JC    S45a;
      A     #InpAlarmNxBottleNotEmpty;
      L     B#(1, 14);	//Message Error ('fault next bottle not empty')
      JC    S45a;
      A     #InpAlarmCoverNotClosed;
      L     B#(1, 15);	//Message Error ('fault cover not closed')
      JC    S45a;
      A     #InpAlarmMultiple;
      L     B#(1, 16);	//Message Error ('fault multiple')
      JC    S45a;
      A     #OutReadingFaultRFID;	//[7.0]
      A     #Par.ParTagReader;	//[7.0]
      L     B#(1, 18);	//[7.0] Message Error ('fault reading RFID')
      JC    S45a;
      A     #StSampling;
      L     B#(1, 10);	//Message Error ('fault sampling')
      JC    S45a;
      L     B#(1, 13);	//Message Error ('fault bottle change')
S45a: T     #tmpLOGvalue;
      R     #StSampling;
      R     #StBottleChange;
      R     #CmdSample;	//Reset commands 
      R     #CmdBottleChange;
      A     #OutResponseFault;	//Condition for StFault
      O     #tmpFault;
      AN    #InWarningMode;	//StXxx -> StFault transition flag
      AN    #tmpLocal;
      JCN   S4J3;
      S     "GCS7_Gr_InFaultFlag";	//Gr.InFaultFlag
      S     #StFault;
      CALL  "SYS_Horn_Code" (
           FcCode                   := 1,
           ParObjectType            := 1029,
           ParObjectNo              := #Par.ParObjectNo,
           ParHornCode              := #Par.ParHornCode);
      L     #tmpLOGvalue;
      JU    LOG;
S4J3: S     #StWarning;
      JU    LOG;	//Condition for StWarning
//=== Logic ====
// If there's a collective alarm it is not allowed to change the bottle, 
// reset fault first, then set bottle change.
//S4:   U     #CmdBottleChange; // 3.0: Allow bottle change if
//      U     #OutCurBottleFull; // 3.0:  alarm current bottle full
//      S     #StWait; // 3.0: --> StWait
//      R     #StFault; 
//      R     #StWarning; 
//    R     #OutResponseFault; 
//    R     #OutResponseTime; 
//  L     B#(3, 9); //Message ('fault cancelled' )
//    SPB   LOG; 
S4:   A     #InLocal;	//Local mode and
      AN    #InManual;	//automatic mode, not manual
      O;
      A     #tmpCmdOk;	//Fault indicated by hardware inputs
      AN    #OutResponseFault;	//not a response fault
      AN    #tmpFault;
      AN    #tmpWarning;
      O;
      AN    #OutResponseFault;	//3.0: Fault reset manually done:
      A     #tmpFaultReset;	//     No InpCmdOk after fault reset
      AN    #tmpFault;
      AN    #tmpWarning;
      O;
      A     #OutSamplerInLocal;	//Sampler in local mode
      AN    #OutResponseFault;	//not a response fault
      AN    #tmpFault;
      AN    #tmpWarning;
      O;
      A     #OutResponseFault;	//Response fault
      A     #tmpFaultReset;
//      S     #StOff                      //[4.2]
      S     #StWait;	//[4.2]
      R     #StFault;
      R     #StWarning;
      R     #OutResponseFault;
      R     #OutResponseTime;
      L     B#(3, 9);	//Message ('fault cancelled' )
      JC    LOG;
      AN    #tmpFaultReset;	//Condition to start timer
      O     #OutResponseTime;
      JC    S4J1;
      S     #OutResponseTime;
      L     #Par.ParAlarmResponseTime;
      T     #Par.OutActResponseTime;
S4J1: AN    #OutResponseTime;
      JC    OUT;
      AN    "GCS7_Gr_OutTick1s";	//Gr.OutTick1S
      L     #Par.OutActResponseTime;
      JC    S4J2;
      +     -10;
      T     #Par.OutActResponseTime;
S4J2: L     0;
      <=I;
      =     #tmpResponseFault;
      R     #OutResponseTime;
      A     #tmpFault;
      O     #tmpWarning;
      A     #tmpResponseFault;	// 3.0:
      L     B#(1, 17);	// 3.0: reLOG Message Error ('alarm reset fault')
      JC    LOG;
      JU    OUT;
NETWORK
TITLE = LOG
LOG:  A     #Par.ParLogOff;	//---Set LOG Message
      JC    OUT;
      T     #tmpLOGvalue;
      L     W#16#FF;
      AW;
      T     #OutAlarmNrLog;
      CALL  "GCS7_LogConvert" (
           ObjectNo                 := #Par.ParObjectNo,
           MsgType                  := #Par.ParMsgType,
           ClassMsgTxt              := #tmpLOGvalue,
           OType                    := 1029);	//LOG Message Converter / Entry / Contains Class and TextNo
NETWORK
TITLE = Global End
//===Handle dyn.OutLocalMode
OUT:  A     #InpSamplerInAuto;
      R     #OutSamplerInLocal;
      AN    #InLocal;
      AN    #InpSamplerInAuto;
      AN    #OutSamplerInLocal;
      S     #OutSamplerInLocal;
      JC    LOM;
      JU    OUTx;
LOM:  AN    #tmpReport;
      JC    OUT;
      L     B#(4, 4);	//Message Info ('sampler in local mode')
      JU    LOG;
//===Set digital outputs
//---OutpAlarmReset
OUTx: A     #StWarning;
      O     #StFault;
      A     #OutResponseTime;
      AN    #OutResponseFault;
      AN    #tmpCmdOk;
      O     #CmdFaultReset;
      AN    "GCS7_Gr_OutTick500ms";
      S     #OutpAlarmReset;
      R     #CmdFaultReset;
      A     "GCS7_Gr_OutTick500ms";
      ON    #InpAlarmCollect;
      R     #OutpAlarmReset;
//---OutpTakeSample
      A     #StSampling;
      =     #OutpSampling;
//---OutpBottleChange
      A     #StBottleChange;
      =     #OutpBottleChange;
//---OutpFunctionRelease
      AN    #InLocal;
      O     #InManual;
      A     #InpSamplerInAuto;
      =     #OutpFuncRelease;
//===Clear Commands and auxiliary signals
//---By not output function release
      AN    #OutpFuncRelease;
      O     #StOff;
      R     #OutCurBottleFull;
      R     #CmdSample;
      R     #CmdBottleChange;
//---All others
      CLR;
      =     #CmdNewBatch;
//---By no product flow
      AN    #InProductFlow;
      A     #OutDelayFault;
      R     #OutProductFlow;
      R     #OutDelayFault;
      R     #CmdSample;
      JCN   STC0;
//[5.2]      L     0
//[5.2]      T     #OutActSampleTime
//[5.2]      T     #OutActBottleChangeTime
//--Output for group 
STC0: AN    #InLocal;
      O     #InManual;
      A     #InDPFault;
      S     "GCS7_Gr_InDPFault";
      AN    #InLocal;
      O     #InManual;
      A     #InHWStop;
      S     "GCS7_Gr_InHWStop";
NETWORK
TITLE = Registering Tag
      NOP   0;
//Resulting Tag
      A     #Tag.HskRead.F_Result;	//[6.2]
      JC    rgJ3;	//[6.2]
      AN    #CmdSendResult;
      O     #Tag.OutRegistrated;
      JC    rgJ1;
      L     #Tag.InJobNr;
      T     #Tag.OutJobNrResult;
      L     #Tag.InBatchNr;
      T     #Tag.OutBatchNrResult;
      L     #Tag.OutTagNrAc;
      T     #Tag.OutTagNrResult;
      SET;
      S     #Tag.HskRead.F_Result;
rgJ1: R     #CmdSendResult;
rgJ3: NOP   0;	//[6.2]
//--------------------------
      AN    #Tag.HskWrite.Q_Result;
      JC    rgJ2;
      L     #Tag.OutTagNrAc;
      L     #Tag.OutTagNrResult;
      ==D;
      A     #Tag.HskRead.F_Result;
      A     #Tag.HskWrite.Q_Result;
      S     #Tag.OutRegistrated;
      SET;
      R     #Tag.HskWrite.Q_Result;
      R     #Tag.HskRead.F_Result;
rgJ2: NOP   0;
//--------------------------
//Init Registered
      L     0;
      L     #Tag.OutTagNrAc;
      <>D;
      A(;
      L     #Tag.OutTagNrResult;
      <>D;
      );
      R     #Tag.OutRegistrated;
NETWORK
TITLE = State Code
      L     1;	//Code: StOff
      A     #StOff;
      JC    STCH;
      L     2;	//Code: StWait
      A     #StWait;
      JC    STC;
      L     3;	//Code: StSampling
      A     #StSampling;
      JC    STC;
      L     4;	//Code: StBottleChange
      A     #StBottleChange;
      JC    STC;
      L     5;	//Code: StWarning
      A     #StWarning;
      JC    STCH;
      L     32;	//Code: StFault
      JU    STC;
//Add +40 if HWStop
STCH: AN    #InHWStop;
      JC    STCD;
      +     40;
      JC    STC;
//Add +50 if DPFault
STCD: AN    #InDPFault;
      JC    STC;
      +     50;
      JC    STC;
STC:  L     #StCode;	//Old state code
      TAK;
      T     #StCode;	//Save state code
      <>I;
      L     3;	//Load code for CBit methode
      CC    "SYS_CBitCtrl";
NETWORK
TITLE = Write Data to Profibus DP
      AN    #Par.ParDP;
      O     #InDPFault;	//[7.0]
      JC    wrJ0;
      LAR1  P##tmpIO;
      L     0;
      T     LD [AR1,P#0.0];
      A     #OutpBottleChange;
      =     #tmpIO.AE33_0;
      A     #OutpSampling;
      =     #tmpIO.AE33_1;
      A     #OutpAlarmReset;
      =     #tmpIO.AE33_2;
      SET;
      =     #tmpIO.AE33_6;
      L     #InSamplePulseLength;
      T     #tmpIO.EAW102;
      LAR1  P##tmpIO;
      L     LD [AR1,P#0.0];
      LAR1  #tmpAddrDP;
      AN    #InSimulation;	//[7.0]
      JC    wrJ1;	//[7.0]
      T     QD [AR1,P#0.0];	//[7.0]
      JC    wrJ0;	//[7.0]
wrJ1: T     PQD [AR1,P#0.0];
wrJ0: NOP   0;
NETWORK
TITLE = [7.0]: Communication RFID
      AN    #Par.ParTagReader;
      BEC;
      L     #Par.ParDBNoRFID;
      T     #tmpDBTagReader;
      OPN   DB [#tmpDBTagReader];
      CDB;
      UC    "SSA_EL_Sampler_RFID";	//Call Tag Reader Baumer
      CDB;
//Data from RFID
      L     DBD 424;	//ToBuhler.OutTagNoAct
      T     #Tag.OutTagNrAc;
      A     DBX 420.0;	//ToBuhler.OutReadingFault
      =     #OutReadingFaultRFID;
//Data To RFID
      A     #tmpFaultReset;
      S     DBX 410.2;	//FromBuhler.CmdFaultReset
      A     #OutBottleInPosition;
      =     DBX 410.0;	//FromBuhler.BottleInPosition
      A     #StBottleChange;
      =     DBX 410.1;	//FromBuhler.StBottleChange
      A     #InSimulation;	//[7.2]
      =     DBX 410.4;	//[7.2] FromBuhler.InSimulation
END_FUNCTION_BLOCK

